KUKA KRL program: ps_a_stb_res_c02.src, ps_a_stb_res_c02.dat

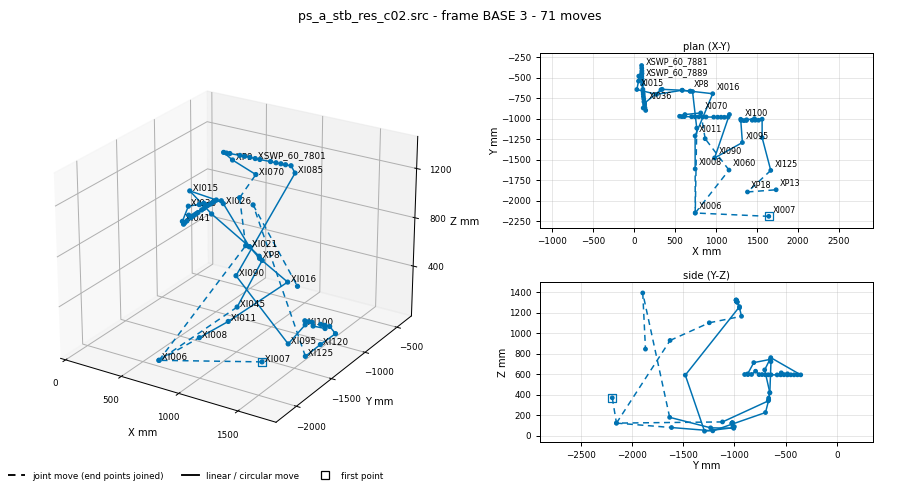
[picture p0: tool path of ps_a_stb_res_c02.src in frame BASE 3, 71 of 71 moves have a stored position in this frame; points joined in program order, loops and branches not executed]
--- ps_a_stb_res_c02.src ---
&ACCESS RVO1
&REL 230
&COMMENT Solda Atego STB
&PARAM DISKPATH = KRC:\R1\Program\OLP
DEF ps_a_stb_res_c02( )

;FOLD INI
;FOLD SPOTTECH INI
USERSPOT(#INIT)
;ENDFOLD (SPOTTECH INI)
;FOLD GRIPPERTECH INI
USER_GRP(0,DUMMY,DUMMY,GDEFAULT)
;ENDFOLD (GRIPPERTECH INI)
  ;FOLD USER INI
    ;Make your modifications here

  ;ENDFOLD (USER INI)
;ENDFOLD (INI)

; Caracterizacao dos meios de producao
; Changes: Solda Respot - ATEGO - STB
; Versao Atual: 18/02/2016
; Ferramenta: Gun C02
; Name: P13.060-R1

chk_w3_wechs_ok ( )              ; CHECK C2

IF (NOT(GHOST())) THEN
IF MaxStandMenge(3) THEN
  MaxStandmengeErreicht(3)
ENDIF
IF Elektrodenwechsel(3) THEN
  e_Fraes_3 ()
ENDIF
ENDIF

;FOLD PTP l007 Vel=100 % P_OLP7 Tool[3]:GUN C2 Base[3]:Atego/Axor;%{PE}%R 8.2.20,%MKUKATPBASIS,%CMOVE,%VPTP,%P 1:PTP, 2:l007, 3:, 5:100, 7:P_OLP7
$BWDSTART=FALSE
PDAT_ACT=PP_OLP7
FDAT_ACT=Fl007
BAS(#PTP_PARAMS,100)
PTP Xl007
;ENDFOLD
;FOLD PTP l006 Vel=100 % P_OLP6 Tool[3]:Gun C02 Base[3]:Atego/Axor;%{PE}%R 8.2.20,%MKUKATPBASIS,%CMOVE,%VPTP,%P 1:PTP, 2:l006, 3:, 5:100, 7:P_OLP6
$BWDSTART=FALSE
PDAT_ACT=PP_OLP6
FDAT_ACT=Fl006
BAS(#PTP_PARAMS,100)
PTP Xl006
;ENDFOLD

;FOLD OUT 3380 'Perfil Livre Estacao' State=TRUE ;%{PE}%R 8.2.20,%MKUKATPBASIS,%COUT,%VOUTX,%P 2:3380, 3:Perfil Livre Estacao, 5:TRUE, 6:
$OUT[3380]=TRUE
;ENDFOLD
;FOLD WAIT FOR ( IN 3380 'Liberacao de Solda' );%{PE}%R 8.2.20,%MKUKATPBASIS,%CEXT_WAIT_FOR,%VEXT_WAIT_FOR,%P 2:, 4:, 5:$IN, 6:3380, 7:Liberacao de Solda, 9:
WAIT FOR  ( $IN[3380] )
;ENDFOLD
;FOLD OUT 3380 'Perfil Livre Estacao' State=FALSE ;%{PE}%R 8.2.20,%MKUKATPBASIS,%COUT,%VOUTX,%P 2:3380, 3:Perfil Livre Estacao, 5:FALSE, 6:
$OUT[3380]=FALSE
;ENDFOLD

;FOLD ; Liga intertravamento 4 com R4;%{PE}%R 8.2.20,%MKUKATPBASIS,%CCOMMENT,%VNORMAL,%P 2:Liga  intertravamento  4  com  R4
;ENDFOLD
;FOLD Collision.Monitoring_4_On ;%{PE}%MKUKATPUSER
COLLSTOP( 4, 1 ) ;Interrupt-Controlled
;ENDFOLD

;FOLD ; Liga intertravamento 10 com R3;%{PE}%R 8.2.20,%MKUKATPBASIS,%CCOMMENT,%VNORMAL,%P 2:Liga  intertravamento  10  com  R3
;ENDFOLD
;FOLD Collision.Monitoring_10_On ;%{PE}%MKUKATPUSER
COLLSTOP( 10, 1 ) ;not Interrupt-Controlled
;ENDFOLD

;FOLD ; Liga intertravamento 5 com R5;%{PE}%R 8.2.20,%MKUKATPBASIS,%CCOMMENT,%VNORMAL,%P 2:Liga  intertravamento  5  com  R5
;ENDFOLD
;FOLD Collision.Monitoring_5_On ;%{PE}%MKUKATPUSER
COLLSTOP( 5, 1 ) ;not Interrupt-Controlled
;ENDFOLD

;FOLD ; Liga intertravamento 12 com R5;%{PE}%R 8.2.20,%MKUKATPBASIS,%CCOMMENT,%VNORMAL,%P 2:Liga  intertravamento  12  com  R5
;ENDFOLD
;FOLD Collision.Monitoring_12_On ;%{PE}%MKUKATPUSER
COLLSTOP( 12, 1 ) ;not Interrupt-Controlled
;ENDFOLD

;FOLD ; Liga intertravamento 13 com R5;%{PE}%R 8.2.20,%MKUKATPBASIS,%CCOMMENT,%VNORMAL,%P 2:Liga  intertravamento  13  com  R5
;ENDFOLD
;FOLD Collision.Monitoring_13_On ;%{PE}%MKUKATPUSER
COLLSTOP( 13, 1 ) ;not Interrupt-Controlled
;ENDFOLD

;FOLD PTP l008 CONT Vel=100 % P_OLP8 Tool[3]:GUN C2 Base[3]:Atego/Axor;%{PE}%R 8.2.20,%MKUKATPBASIS,%CMOVE,%VPTP,%P 1:PTP, 2:l008, 3:C_DIS, 5:100, 7:P_OLP8
$BWDSTART=FALSE
PDAT_ACT=PP_OLP8
FDAT_ACT=Fl008
BAS(#PTP_PARAMS,100)
PTP Xl008 C_DIS
;ENDFOLD
;FOLD LIN l011 CONT Vel=2 m/s L_OLP42 Tool[3]:GUN C2 Base[3]:Atego/Axor;%{PE}%R 8.2.20,%MKUKATPBASIS,%CMOVE,%VLIN,%P 1:LIN, 2:l011, 3:C_DIS C_DIS, 5:2, 7:L_OLP42
$BWDSTART=FALSE
LDAT_ACT=LL_OLP42
FDAT_ACT=Fl011
BAS(#CP_PARAMS,2)
LIN Xl011 C_DIS C_DIS
;ENDFOLD
;FOLD LIN l016 CONT Vel=2 m/s CPDAT11 Tool[3]:GUN C2 Base[3]:Atego/Axor;%{PE}%R 8.2.20,%MKUKATPBASIS,%CMOVE,%VLIN,%P 1:LIN, 2:l016, 3:C_DIS C_DIS, 5:2, 7:CPDAT11
$BWDSTART=FALSE
LDAT_ACT=LCPDAT11
FDAT_ACT=Fl016
BAS(#CP_PARAMS,2)
LIN Xl016 C_DIS C_DIS
;ENDFOLD
;FOLD LIN P8 CONT Vel=2 m/s CPDAT8 Tool[3]:GUN C2 Base[3]:Atego/Axor;%{PE}%R 8.2.20,%MKUKATPBASIS,%CMOVE,%VLIN,%P 1:LIN, 2:P8, 3:C_DIS C_DIS, 5:2, 7:CPDAT8
$BWDSTART=FALSE
LDAT_ACT=LCPDAT8
FDAT_ACT=FP8
BAS(#CP_PARAMS,2)
LIN XP8 C_DIS C_DIS
;ENDFOLD
;FOLD LIN l021 CONT Vel=2 m/s L_OLP44 Tool[3]:GUN C2 Base[3]:Atego/Axor;%{PE}%R 8.2.20,%MKUKATPBASIS,%CMOVE,%VLIN,%P 1:LIN, 2:l021, 3:C_DIS C_DIS, 5:2, 7:L_OLP44
$BWDSTART=FALSE
LDAT_ACT=LL_OLP44
FDAT_ACT=Fl021
BAS(#CP_PARAMS,2)
LIN Xl021 C_DIS C_DIS
;ENDFOLD
;FOLD LIN l026 CONT Vel=2 m/s L_OLP45 Tool[3]:GUN C2 Base[3]:Atego/Axor;%{PE}%R 8.2.20,%MKUKATPBASIS,%CMOVE,%VLIN,%P 1:LIN, 2:l026, 3:C_DIS C_DIS, 5:2, 7:L_OLP45
$BWDSTART=FALSE
LDAT_ACT=LL_OLP45
FDAT_ACT=Fl026
BAS(#CP_PARAMS,2)
LIN Xl026 C_DIS C_DIS
;ENDFOLD
;FOLD LIN l031 CONT Vel=1 m/s L_OLP46 Tool[3]:GUN C2 Base[3]:Atego/Axor;%{PE}%R 8.2.20,%MKUKATPBASIS,%CMOVE,%VLIN,%P 1:LIN, 2:l031, 3:C_DIS C_DIS, 5:1, 7:L_OLP46
$BWDSTART=FALSE
LDAT_ACT=LL_OLP46
FDAT_ACT=Fl031
BAS(#CP_PARAMS,1)
LIN Xl031 C_DIS C_DIS
;ENDFOLD
;FOLD LIN l036 CONT Vel=2 m/s L_OLP47 Tool[3]:GUN C2 Base[3]:Atego/Axor;%{PE}%R 8.2.20,%MKUKATPBASIS,%CMOVE,%VLIN,%P 1:LIN, 2:l036, 3:C_DIS C_DIS, 5:2, 7:L_OLP47
$BWDSTART=FALSE
LDAT_ACT=LL_OLP47
FDAT_ACT=Fl036
BAS(#CP_PARAMS,2)
LIN Xl036 C_DIS C_DIS
;ENDFOLD
;FOLD LIN l041 CONT Vel=2 m/s L_OLP48 Tool[3]:GUN C2 Base[3]:Atego/Axor;%{PE}%R 8.2.20,%MKUKATPBASIS,%CMOVE,%VLIN,%P 1:LIN, 2:l041, 3:C_DIS C_DIS, 5:2, 7:L_OLP48
$BWDSTART=FALSE
LDAT_ACT=LL_OLP48
FDAT_ACT=Fl041
BAS(#CP_PARAMS,2)
LIN Xl041 C_DIS C_DIS
;ENDFOLD

;FOLD ; SWP_60_7345;%{PE}%R 8.2.20,%MKUKATPBASIS,%CCOMMENT,%VNORMAL,%P 2:SWP_60_7345
;ENDFOLD
;FOLD LIN swp_60_7345 CPDAT13 SPOT Gun=2 RETR CLS PgNo1=186 ACTIVE=1 Tool[3]:GUN C2 Base[3]:Atego/Axor;%{PE}%R 8.2.2,%MKUKATPSPOT,%CSPOT,%VLIN,%P 1:LIN, 2:swp_60_7345, 3:, 5:2, 7:CPDAT13, 10:2, 12:#FIRST, 14:#CLO, 16:186, 18:1, 20:0, 22:0, 24:1, 25:NORMAL
$BWDSTART=FALSE
LDAT_ACT=LCPDAT13
FDAT_ACT=Fswp_60_7345
BAS(#CP_PARAMS,LCPDAT13.VEL)
S_ACT.GUN=2
S_ACT.PAIR=SDEFAULT.PAIR
S_ACT.RETR=#CLO
S_ACT.CLO_TM=1
S_ACT.PGNO1=186
S_ACT.PGNO2=SDEFAULT.PGNO2
S_ACT.PRESS1=SDEFAULT.PRESS1
S_ACT.PRESS2=SDEFAULT.PRESS2
S_READY=FALSE
LIN Xswp_60_7345
USERSPOT(#SPOT, S_ACT)
WAIT FOR S_READY
;ENDFOLD

;FOLD ; SWP_60_7909;%{PE}%R 8.2.20,%MKUKATPBASIS,%CCOMMENT,%VNORMAL,%P 2:SWP_60_7909
;ENDFOLD
;FOLD LIN SWP_60_7909 L_OLP49 SPOT Gun=2 RETR CLS PgNo1=186 ACTIVE=1 Tool[3]:GUN C2 Base[3]:Atego/Axor;%{PE}%R 8.2.2,%MKUKATPSPOT,%CSPOT,%VLIN,%P 1:LIN, 2:SWP_60_7909, 3:, 5:2, 7:L_OLP49, 10:2, 12:#FIRST, 14:#CLO, 16:186, 18:1, 20:0, 22:0, 24:1, 25:NORMAL
$BWDSTART=FALSE
LDAT_ACT=LL_OLP49
FDAT_ACT=FSWP_60_7909
BAS(#CP_PARAMS,LL_OLP49.VEL)
S_ACT.GUN=2
S_ACT.PAIR=SDEFAULT.PAIR
S_ACT.RETR=#CLO
S_ACT.CLO_TM=1
S_ACT.PGNO1=186
S_ACT.PGNO2=SDEFAULT.PGNO2
S_ACT.PRESS1=SDEFAULT.PRESS1
S_ACT.PRESS2=SDEFAULT.PRESS2
S_READY=FALSE
LIN XSWP_60_7909
USERSPOT(#SPOT, S_ACT)
WAIT FOR S_READY
;ENDFOLD

;FOLD ; SWP_60_7907;%{PE}%R 8.2.20,%MKUKATPBASIS,%CCOMMENT,%VNORMAL,%P 2:SWP_60_7907
;ENDFOLD
;FOLD LIN SWP_60_7907 CPDAT1 SPOT Gun=2 RETR CLS PgNo1=186 ACTIVE=1 Tool[3]:GUN C2 Base[3]:Atego/Axor;%{PE}%R 8.2.2,%MKUKATPSPOT,%CSPOT,%VLIN,%P 1:LIN, 2:SWP_60_7907, 3:, 5:0.001, 7:CPDAT1, 10:2, 12:#FIRST, 14:#CLO, 16:186, 18:1, 20:0, 22:0, 24:1, 25:NORMAL
$BWDSTART=FALSE
LDAT_ACT=LCPDAT1
FDAT_ACT=FSWP_60_7907
BAS(#CP_PARAMS,LCPDAT1.VEL)
S_ACT.GUN=2
S_ACT.PAIR=SDEFAULT.PAIR
S_ACT.RETR=#CLO
S_ACT.CLO_TM=1
S_ACT.PGNO1=186
S_ACT.PGNO2=SDEFAULT.PGNO2
S_ACT.PRESS1=SDEFAULT.PRESS1
S_ACT.PRESS2=SDEFAULT.PRESS2
S_READY=FALSE
LIN XSWP_60_7907
USERSPOT(#SPOT, S_ACT)
WAIT FOR S_READY
;ENDFOLD

;FOLD LIN l042 CONT Vel=2 m/s L_OLP65 Tool[3]:GUN C2 Base[3]:Atego/Axor;%{PE}%R 8.2.20,%MKUKATPBASIS,%CMOVE,%VLIN,%P 1:LIN, 2:l042, 3:C_DIS C_DIS, 5:2, 7:L_OLP65
$BWDSTART=FALSE
LDAT_ACT=LL_OLP65
FDAT_ACT=Fl042
BAS(#CP_PARAMS,2)
LIN Xl042 C_DIS C_DIS
;ENDFOLD

;FOLD ; SWP_60_7905;%{PE}%R 8.2.20,%MKUKATPBASIS,%CCOMMENT,%VNORMAL,%P 2:SWP_60_7905
;ENDFOLD
;FOLD LIN SWP_60_7905 L_OLP51 SPOT Gun=2 RETR CLS PgNo1=186 ACTIVE=1 Tool[3]:GUN C2 Base[3]:Atego/Axor;%{PE}%R 8.2.2,%MKUKATPSPOT,%CSPOT,%VLIN,%P 1:LIN, 2:SWP_60_7905, 3:, 5:2, 7:L_OLP51, 10:2, 12:#FIRST, 14:#CLO, 16:186, 18:1, 20:0, 22:0, 24:1, 25:NORMAL
$BWDSTART=FALSE
LDAT_ACT=LL_OLP51
FDAT_ACT=FSWP_60_7905
BAS(#CP_PARAMS,LL_OLP51.VEL)
S_ACT.GUN=2
S_ACT.PAIR=SDEFAULT.PAIR
S_ACT.RETR=#CLO
S_ACT.CLO_TM=1
S_ACT.PGNO1=186
S_ACT.PGNO2=SDEFAULT.PGNO2
S_ACT.PRESS1=SDEFAULT.PRESS1
S_ACT.PRESS2=SDEFAULT.PRESS2
S_READY=FALSE
LIN XSWP_60_7905
USERSPOT(#SPOT, S_ACT)
WAIT FOR S_READY
;ENDFOLD

;FOLD ; SWP_60_7903;%{PE}%R 8.2.20,%MKUKATPBASIS,%CCOMMENT,%VNORMAL,%P 2:SWP_60_7903
;ENDFOLD
;FOLD LIN SWP_60_7903 L_OLP52 SPOT Gun=2 RETR CLS PgNo1=186 ACTIVE=1 Tool[3]:GUN C2 Base[3]:Atego/Axor;%{PE}%R 8.2.2,%MKUKATPSPOT,%CSPOT,%VLIN,%P 1:LIN, 2:SWP_60_7903, 3:, 5:2, 7:L_OLP52, 10:2, 12:#FIRST, 14:#CLO, 16:186, 18:1, 20:0, 22:0, 24:1, 25:NORMAL
$BWDSTART=FALSE
LDAT_ACT=LL_OLP52
FDAT_ACT=FSWP_60_7903
BAS(#CP_PARAMS,LL_OLP52.VEL)
S_ACT.GUN=2
S_ACT.PAIR=SDEFAULT.PAIR
S_ACT.RETR=#CLO
S_ACT.CLO_TM=1
S_ACT.PGNO1=186
S_ACT.PGNO2=SDEFAULT.PGNO2
S_ACT.PRESS1=SDEFAULT.PRESS1
S_ACT.PRESS2=SDEFAULT.PRESS2
S_READY=FALSE
LIN XSWP_60_7903
USERSPOT(#SPOT, S_ACT)
WAIT FOR S_READY
;ENDFOLD

;FOLD ; SWP_60_7901;%{PE}%R 8.2.20,%MKUKATPBASIS,%CCOMMENT,%VNORMAL,%P 2:SWP_60_7901
;ENDFOLD
;FOLD LIN SWP_60_7901 L_OLP53 SPOT Gun=2 RETR CLS PgNo1=186 ACTIVE=1 Tool[3]:GUN C2 Base[3]:Atego/Axor;%{PE}%R 8.2.2,%MKUKATPSPOT,%CSPOT,%VLIN,%P 1:LIN, 2:SWP_60_7901, 3:, 5:2, 7:L_OLP53, 10:2, 12:#FIRST, 14:#CLO, 16:186, 18:1, 20:0, 22:0, 24:1, 25:NORMAL
$BWDSTART=FALSE
LDAT_ACT=LL_OLP53
FDAT_ACT=FSWP_60_7901
BAS(#CP_PARAMS,LL_OLP53.VEL)
S_ACT.GUN=2
S_ACT.PAIR=SDEFAULT.PAIR
S_ACT.RETR=#CLO
S_ACT.CLO_TM=1
S_ACT.PGNO1=186
S_ACT.PGNO2=SDEFAULT.PGNO2
S_ACT.PRESS1=SDEFAULT.PRESS1
S_ACT.PRESS2=SDEFAULT.PRESS2
S_READY=FALSE
LIN XSWP_60_7901
USERSPOT(#SPOT, S_ACT)
WAIT FOR S_READY
;ENDFOLD

;FOLD ; SWP_60_7329;%{PE}%R 8.2.20,%MKUKATPBASIS,%CCOMMENT,%VNORMAL,%P 2:SWP_60_7329
;ENDFOLD
;FOLD LIN SWP_60_7329 L_OLP54 SPOT Gun=2 RETR CLS PgNo1=186 ACTIVE=1 Tool[3]:GUN C2 Base[3]:Atego/Axor;%{PE}%R 8.2.2,%MKUKATPSPOT,%CSPOT,%VLIN,%P 1:LIN, 2:SWP_60_7329, 3:, 5:2, 7:L_OLP54, 10:2, 12:#FIRST, 14:#CLO, 16:186, 18:1, 20:0, 22:0, 24:1, 25:NORMAL
$BWDSTART=FALSE
LDAT_ACT=LL_OLP54
FDAT_ACT=FSWP_60_7329
BAS(#CP_PARAMS,LL_OLP54.VEL)
S_ACT.GUN=2
S_ACT.PAIR=SDEFAULT.PAIR
S_ACT.RETR=#CLO
S_ACT.CLO_TM=1
S_ACT.PGNO1=186
S_ACT.PGNO2=SDEFAULT.PGNO2
S_ACT.PRESS1=SDEFAULT.PRESS1
S_ACT.PRESS2=SDEFAULT.PRESS2
S_READY=FALSE
LIN XSWP_60_7329
USERSPOT(#SPOT, S_ACT)
WAIT FOR S_READY
;ENDFOLD

;FOLD ; SWP_60_7897;%{PE}%R 8.2.20,%MKUKATPBASIS,%CCOMMENT,%VNORMAL,%P 2:SWP_60_7897
;ENDFOLD
;FOLD LIN SWP_60_7897 CPDAT14 SPOT Gun=2 RETR CLS PgNo1=186 ACTIVE=1 Tool[3]:GUN C2 Base[3]:Atego/Axor;%{PE}%R 8.2.2,%MKUKATPSPOT,%CSPOT,%VLIN,%P 1:LIN, 2:SWP_60_7897, 3:, 5:2, 7:CPDAT14, 10:2, 12:#FIRST, 14:#CLO, 16:186, 18:1, 20:0, 22:0, 24:1, 25:NORMAL
$BWDSTART=FALSE
LDAT_ACT=LCPDAT14
FDAT_ACT=FSWP_60_7897
BAS(#CP_PARAMS,LCPDAT14.VEL)
S_ACT.GUN=2
S_ACT.PAIR=SDEFAULT.PAIR
S_ACT.RETR=#CLO
S_ACT.CLO_TM=1
S_ACT.PGNO1=186
S_ACT.PGNO2=SDEFAULT.PGNO2
S_ACT.PRESS1=SDEFAULT.PRESS1
S_ACT.PRESS2=SDEFAULT.PRESS2
S_READY=FALSE
LIN XSWP_60_7897
USERSPOT(#SPOT, S_ACT)
WAIT FOR S_READY
;ENDFOLD

;FOLD ; SWP_60_7893;%{PE}%R 8.2.20,%MKUKATPBASIS,%CCOMMENT,%VNORMAL,%P 2:SWP_60_7893
;ENDFOLD
;FOLD LIN SWP_60_7893 L_OLP55 SPOT Gun=2 RETR CLS PgNo1=186 ACTIVE=1 Tool[3]:GUN C2 Base[3]:Atego/Axor;%{PE}%R 8.2.2,%MKUKATPSPOT,%CSPOT,%VLIN,%P 1:LIN, 2:SWP_60_7893, 3:, 5:2, 7:L_OLP55, 10:2, 12:#FIRST, 14:#CLO, 16:186, 18:1, 20:0, 22:0, 24:1, 25:NORMAL
$BWDSTART=FALSE
LDAT_ACT=LL_OLP55
FDAT_ACT=FSWP_60_7893
BAS(#CP_PARAMS,LL_OLP55.VEL)
S_ACT.GUN=2
S_ACT.PAIR=SDEFAULT.PAIR
S_ACT.RETR=#CLO
S_ACT.CLO_TM=1
S_ACT.PGNO1=186
S_ACT.PGNO2=SDEFAULT.PGNO2
S_ACT.PRESS1=SDEFAULT.PRESS1
S_ACT.PRESS2=SDEFAULT.PRESS2
S_READY=FALSE
LIN XSWP_60_7893
USERSPOT(#SPOT, S_ACT)
WAIT FOR S_READY
;ENDFOLD

;FOLD ; SWP_60_7891;%{PE}%R 8.2.20,%MKUKATPBASIS,%CCOMMENT,%VNORMAL,%P 2:SWP_60_7891
;ENDFOLD
;FOLD LIN SWP_60_7891 L_OLP56 SPOT Gun=2 RETR CLS PgNo1=186 ACTIVE=1 Tool[3]:GUN C2 Base[3]:Atego/Axor;%{PE}%R 8.2.2,%MKUKATPSPOT,%CSPOT,%VLIN,%P 1:LIN, 2:SWP_60_7891, 3:, 5:2, 7:L_OLP56, 10:2, 12:#FIRST, 14:#CLO, 16:186, 18:1, 20:0, 22:0, 24:1, 25:NORMAL
$BWDSTART=FALSE
LDAT_ACT=LL_OLP56
FDAT_ACT=FSWP_60_7891
BAS(#CP_PARAMS,LL_OLP56.VEL)
S_ACT.GUN=2
S_ACT.PAIR=SDEFAULT.PAIR
S_ACT.RETR=#CLO
S_ACT.CLO_TM=1
S_ACT.PGNO1=186
S_ACT.PGNO2=SDEFAULT.PGNO2
S_ACT.PRESS1=SDEFAULT.PRESS1
S_ACT.PRESS2=SDEFAULT.PRESS2
S_READY=FALSE
LIN XSWP_60_7891
USERSPOT(#SPOT, S_ACT)
WAIT FOR S_READY
;ENDFOLD

;FOLD ; SWP_60_7889;%{PE}%R 8.2.20,%MKUKATPBASIS,%CCOMMENT,%VNORMAL,%P 2:SWP_60_7889
;ENDFOLD
;FOLD LIN SWP_60_7889 L_OLP57 SPOT Gun=2 RETR OPN PgNo1=186 ACTIVE=1 Tool[3]:GUN C2 Base[3]:Atego/Axor;%{PE}%R 8.2.2,%MKUKATPSPOT,%CSPOT,%VLIN,%P 1:LIN, 2:SWP_60_7889, 3:, 5:2, 7:L_OLP57, 10:2, 12:#FIRST, 14:#OPN, 16:186, 18:1, 20:0, 22:0, 24:1, 25:NORMAL
$BWDSTART=FALSE
LDAT_ACT=LL_OLP57
FDAT_ACT=FSWP_60_7889
BAS(#CP_PARAMS,LL_OLP57.VEL)
S_ACT.GUN=2
S_ACT.PAIR=SDEFAULT.PAIR
S_ACT.RETR=#OPN
S_ACT.CLO_TM=1
S_ACT.PGNO1=186
S_ACT.PGNO2=SDEFAULT.PGNO2
S_ACT.PRESS1=SDEFAULT.PRESS1
S_ACT.PRESS2=SDEFAULT.PRESS2
S_READY=FALSE
LIN XSWP_60_7889
USERSPOT(#SPOT, S_ACT)
WAIT FOR S_READY
;ENDFOLD

;FOLD LIN P4 CONT Vel=1 m/s CPDAT4 Tool[3]:GUN C2 Base[3]:Atego/Axor;%{PE}%R 8.2.20,%MKUKATPBASIS,%CMOVE,%VLIN,%P 1:LIN, 2:P4, 3:C_DIS C_DIS, 5:1, 7:CPDAT4
$BWDSTART=FALSE
LDAT_ACT=LCPDAT4
FDAT_ACT=FP4
BAS(#CP_PARAMS,1)
LIN XP4 C_DIS C_DIS
;ENDFOLD
;FOLD LIN P5 CONT Vel=1 m/s CPDAT5 Tool[3]:GUN C2 Base[3]:Atego/Axor;%{PE}%R 8.2.20,%MKUKATPBASIS,%CMOVE,%VLIN,%P 1:LIN, 2:P5, 3:C_DIS C_DIS, 5:1, 7:CPDAT5
$BWDSTART=FALSE
LDAT_ACT=LCPDAT5
FDAT_ACT=FP5
BAS(#CP_PARAMS,1)
LIN XP5 C_DIS C_DIS
;ENDFOLD

;FOLD ; SWP_60_7887;%{PE}%R 8.2.20,%MKUKATPBASIS,%CCOMMENT,%VNORMAL,%P 2:SWP_60_7887
;ENDFOLD
;FOLD LIN SWP_60_7887 L_OLP58 SPOT Gun=2 RETR CLS PgNo1=186 ACTIVE=1 Tool[3]:GUN C2 Base[3]:Atego/Axor;%{PE}%R 8.2.2,%MKUKATPSPOT,%CSPOT,%VLIN,%P 1:LIN, 2:SWP_60_7887, 3:, 5:2, 7:L_OLP58, 10:2, 12:#FIRST, 14:#CLO, 16:186, 18:1, 20:0, 22:0, 24:1, 25:NORMAL
$BWDSTART=FALSE
LDAT_ACT=LL_OLP58
FDAT_ACT=FSWP_60_7887
BAS(#CP_PARAMS,LL_OLP58.VEL)
S_ACT.GUN=2
S_ACT.PAIR=SDEFAULT.PAIR
S_ACT.RETR=#CLO
S_ACT.CLO_TM=1
S_ACT.PGNO1=186
S_ACT.PGNO2=SDEFAULT.PGNO2
S_ACT.PRESS1=SDEFAULT.PRESS1
S_ACT.PRESS2=SDEFAULT.PRESS2
S_READY=FALSE
LIN XSWP_60_7887
USERSPOT(#SPOT, S_ACT)
WAIT FOR S_READY
;ENDFOLD

;FOLD ; SWP_60_7885;%{PE}%R 8.2.20,%MKUKATPBASIS,%CCOMMENT,%VNORMAL,%P 2:SWP_60_7885
;ENDFOLD
;FOLD LIN SWP_60_7885 L_OLP59 SPOT Gun=2 RETR CLS PgNo1=186 ACTIVE=1 Tool[3]:GUN C2 Base[3]:Atego/Axor;%{PE}%R 8.2.2,%MKUKATPSPOT,%CSPOT,%VLIN,%P 1:LIN, 2:SWP_60_7885, 3:, 5:2, 7:L_OLP59, 10:2, 12:#FIRST, 14:#CLO, 16:186, 18:1, 20:0, 22:0, 24:1, 25:NORMAL
$BWDSTART=FALSE
LDAT_ACT=LL_OLP59
FDAT_ACT=FSWP_60_7885
BAS(#CP_PARAMS,LL_OLP59.VEL)
S_ACT.GUN=2
S_ACT.PAIR=SDEFAULT.PAIR
S_ACT.RETR=#CLO
S_ACT.CLO_TM=1
S_ACT.PGNO1=186
S_ACT.PGNO2=SDEFAULT.PGNO2
S_ACT.PRESS1=SDEFAULT.PRESS1
S_ACT.PRESS2=SDEFAULT.PRESS2
S_READY=FALSE
LIN XSWP_60_7885
USERSPOT(#SPOT, S_ACT)
WAIT FOR S_READY
;ENDFOLD

;FOLD ; SWP_60_7883;%{PE}%R 8.2.20,%MKUKATPBASIS,%CCOMMENT,%VNORMAL,%P 2:SWP_60_7883
;ENDFOLD
;FOLD LIN SWP_60_7883 L_OLP60 SPOT Gun=2 RETR CLS PgNo1=186 ACTIVE=1 Tool[3]:GUN C2 Base[3]:Atego/Axor;%{PE}%R 8.2.2,%MKUKATPSPOT,%CSPOT,%VLIN,%P 1:LIN, 2:SWP_60_7883, 3:, 5:2, 7:L_OLP60, 10:2, 12:#FIRST, 14:#CLO, 16:186, 18:1, 20:0, 22:0, 24:1, 25:NORMAL
$BWDSTART=FALSE
LDAT_ACT=LL_OLP60
FDAT_ACT=FSWP_60_7883
BAS(#CP_PARAMS,LL_OLP60.VEL)
S_ACT.GUN=2
S_ACT.PAIR=SDEFAULT.PAIR
S_ACT.RETR=#CLO
S_ACT.CLO_TM=1
S_ACT.PGNO1=186
S_ACT.PGNO2=SDEFAULT.PGNO2
S_ACT.PRESS1=SDEFAULT.PRESS1
S_ACT.PRESS2=SDEFAULT.PRESS2
S_READY=FALSE
LIN XSWP_60_7883
USERSPOT(#SPOT, S_ACT)
WAIT FOR S_READY
;ENDFOLD

;FOLD ; SWP_60_7881;%{PE}%R 8.2.20,%MKUKATPBASIS,%CCOMMENT,%VNORMAL,%P 2:SWP_60_7881
;ENDFOLD
;FOLD LIN SWP_60_7881 L_OLP61 SPOT Gun=2 RETR CLS PgNo1=186 ACTIVE=1 Tool[3]:GUN C2 Base[3]:Atego/Axor;%{PE}%R 8.2.2,%MKUKATPSPOT,%CSPOT,%VLIN,%P 1:LIN, 2:SWP_60_7881, 3:, 5:2, 7:L_OLP61, 10:2, 12:#FIRST, 14:#CLO, 16:186, 18:1, 20:0, 22:0, 24:1, 25:NORMAL
$BWDSTART=FALSE
LDAT_ACT=LL_OLP61
FDAT_ACT=FSWP_60_7881
BAS(#CP_PARAMS,LL_OLP61.VEL)
S_ACT.GUN=2
S_ACT.PAIR=SDEFAULT.PAIR
S_ACT.RETR=#CLO
S_ACT.CLO_TM=1
S_ACT.PGNO1=186
S_ACT.PGNO2=SDEFAULT.PGNO2
S_ACT.PRESS1=SDEFAULT.PRESS1
S_ACT.PRESS2=SDEFAULT.PRESS2
S_READY=FALSE
LIN XSWP_60_7881
USERSPOT(#SPOT, S_ACT)
WAIT FOR S_READY
;ENDFOLD

;FOLD ; SWP_60_7311;%{PE}%R 8.2.20,%MKUKATPBASIS,%CCOMMENT,%VNORMAL,%P 2:SWP_60_7311
;ENDFOLD
;FOLD LIN SWP_60_7311 L_OLP48 SPOT Gun=2 RETR CLS PgNo1=186 ACTIVE=1 Tool[3]:GUN C2 Base[3]:Atego/Axor;%{PE}%R 8.2.2,%MKUKATPSPOT,%CSPOT,%VLIN,%P 1:LIN, 2:SWP_60_7311, 3:, 5:2, 7:L_OLP48, 10:2, 12:#FIRST, 14:#CLO, 16:186, 18:1, 20:0, 22:0, 24:1, 25:NORMAL
$BWDSTART=FALSE
LDAT_ACT=LL_OLP48
FDAT_ACT=FSWP_60_7311
BAS(#CP_PARAMS,LL_OLP48.VEL)
S_ACT.GUN=2
S_ACT.PAIR=SDEFAULT.PAIR
S_ACT.RETR=#CLO
S_ACT.CLO_TM=1
S_ACT.PGNO1=186
S_ACT.PGNO2=SDEFAULT.PGNO2
S_ACT.PRESS1=SDEFAULT.PRESS1
S_ACT.PRESS2=SDEFAULT.PRESS2
S_READY=FALSE
LIN XSWP_60_7311
USERSPOT(#SPOT, S_ACT)
WAIT FOR S_READY
;ENDFOLD

;FOLD LIN l015  Vel=2.00 m/s L_OLP3 Tool[3]:GUN C2 Base[3]:Atego/Axor;%{PE}%R8.2.19,%MKUKATPBASIS,%CMOVE,%VLIN,%P 1:LIN, 2:l015, 3: , 5:2.00, 7:L_OLP3
$BWDSTART = FALSE
LDAT_ACT= LL_OLP3
FDAT_ACT= Fl015
BAS(#CP_PARAMS,2.00)
LIN Xl015
;ENDFOLD
;FOLD LIN l030 CONT Vel=2 m/s L_OLP6 Tool[3]:GUN C2 Base[3]:Atego/Axor;%{PE}%R 8.2.20,%MKUKATPBASIS,%CMOVE,%VLIN,%P 1:LIN, 2:l030, 3:C_DIS C_DIS, 5:2, 7:L_OLP6
$BWDSTART=FALSE
LDAT_ACT=LL_OLP6
FDAT_ACT=Fl030
BAS(#CP_PARAMS,2)
LIN Xl030 C_DIS C_DIS
;ENDFOLD
;FOLD LIN l035 CONT Vel=2 m/s L_OLP7 Tool[3]:GUN C2 Base[3]:Atego/Axor;%{PE}%R 8.2.20,%MKUKATPBASIS,%CMOVE,%VLIN,%P 1:LIN, 2:l035, 3:C_DIS C_DIS, 5:2, 7:L_OLP7
$BWDSTART=FALSE
LDAT_ACT=LL_OLP7
FDAT_ACT=Fl035
BAS(#CP_PARAMS,2)
LIN Xl035 C_DIS C_DIS
;ENDFOLD
;FOLD LIN P7 CONT Vel=2 m/s CPDAT7 Tool[3]:GUN C2 Base[3]:Atego/Axor;%{PE}%R 8.2.20,%MKUKATPBASIS,%CMOVE,%VLIN,%P 1:LIN, 2:P7, 3:C_DIS C_DIS, 5:2, 7:CPDAT7
$BWDSTART=FALSE
LDAT_ACT=LCPDAT7
FDAT_ACT=FP7
BAS(#CP_PARAMS,2)
LIN XP7 C_DIS C_DIS
;ENDFOLD
;FOLD LIN l040 CONT Vel=2 m/s L_OLP8 Tool[3]:GUN C2 Base[3]:Atego/Axor;%{PE}%R 8.2.20,%MKUKATPBASIS,%CMOVE,%VLIN,%P 1:LIN, 2:l040, 3:C_DIS C_DIS, 5:2, 7:L_OLP8
$BWDSTART=FALSE
LDAT_ACT=LL_OLP8
FDAT_ACT=Fl040
BAS(#CP_PARAMS,2)
LIN Xl040 C_DIS C_DIS
;ENDFOLD
;FOLD LIN l045 CONT Vel=2 m/s L_OLP9 Tool[3]:GUN C2 Base[3]:Atego/Axor;%{PE}%R 8.2.20,%MKUKATPBASIS,%CMOVE,%VLIN,%P 1:LIN, 2:l045, 3:C_DIS C_DIS, 5:2, 7:L_OLP9
$BWDSTART=FALSE
LDAT_ACT=LL_OLP9
FDAT_ACT=Fl045
BAS(#CP_PARAMS,2)
LIN Xl045 C_DIS C_DIS
;ENDFOLD
;FOLD PTP l050 Vel=100 % PDAT4 Tool[3]:GUN C2 Base[3]:Atego/Axor;%{PE}%R 8.2.20,%MKUKATPBASIS,%CMOVE,%VPTP,%P 1:PTP, 2:l050, 3:, 5:100, 7:PDAT4
$BWDSTART=FALSE
PDAT_ACT=PPDAT4
FDAT_ACT=Fl050
BAS(#PTP_PARAMS,100)
PTP Xl050
;ENDFOLD

;FOLD ; Desliga intertravamento 4 com R4;%{PE}%R 8.2.20,%MKUKATPBASIS,%CCOMMENT,%VNORMAL,%P 2:Desliga  intertravamento  4  com  R4
;ENDFOLD
;FOLD Collision.Monitoring_4_Off . ;%{PE}%MKUKATPUSER
COLLSTOP( 4, 2+0 )
;ENDFOLD

;FOLD ; Desliga intertravamento 10 com R3;%{PE}%R 8.2.20,%MKUKATPBASIS,%CCOMMENT,%VNORMAL,%P 2:Desliga  intertravamento  10  com  R3
;ENDFOLD
;FOLD Collision.Monitoring_10_Off . ;%{PE}%MKUKATPUSER
COLLSTOP( 10, 2+0 )
;ENDFOLD

;FOLD ; Desliga intertravamento 5 com R5;%{PE}%R 8.2.20,%MKUKATPBASIS,%CCOMMENT,%VNORMAL,%P 2:Desliga  intertravamento  5  com  R5
;ENDFOLD
;FOLD Collision.Monitoring_5_Off . ;%{PE}%MKUKATPUSER
COLLSTOP( 5, 2+0 )
;ENDFOLD

;FOLD ; Desliga intertravamento 13 com R5;%{PE}%R 8.2.20,%MKUKATPBASIS,%CCOMMENT,%VNORMAL,%P 2:Desliga  intertravamento  13  com  R5
;ENDFOLD
;FOLD Collision.Monitoring_13_Off . ;%{PE}%MKUKATPUSER
COLLSTOP( 13, 2+0 )
;ENDFOLD

;FOLD PTP l060 CONT Vel=100 % P_OLP2 Tool[3]:GUN C2 Base[3]:Atego/Axor;%{PE}%R 8.2.20,%MKUKATPBASIS,%CMOVE,%VPTP,%P 1:PTP, 2:l060, 3:C_DIS, 5:100, 7:P_OLP2
$BWDSTART=FALSE
PDAT_ACT=PP_OLP2
FDAT_ACT=Fl060
BAS(#PTP_PARAMS,100)
PTP Xl060 C_DIS
;ENDFOLD
;FOLD PTP l065 CONT Vel=100 % P_OLP3 Tool[3]:GUN C2 Base[3]:Atego/Axor;%{PE}%R 8.2.20,%MKUKATPBASIS,%CMOVE,%VPTP,%P 1:PTP, 2:l065, 3:C_DIS, 5:100, 7:P_OLP3
$BWDSTART=FALSE
PDAT_ACT=PP_OLP3
FDAT_ACT=Fl065
BAS(#PTP_PARAMS,100)
PTP Xl065 C_DIS
;ENDFOLD
;FOLD PTP l070 CONT Vel=100 % P_OLP4 Tool[3]:GUN C2 Base[3]:Atego/Axor;%{PE}%R 8.2.20,%MKUKATPBASIS,%CMOVE,%VPTP,%P 1:PTP, 2:l070, 3:C_DIS, 5:100, 7:P_OLP4
$BWDSTART=FALSE
PDAT_ACT=PP_OLP4
FDAT_ACT=Fl070
BAS(#PTP_PARAMS,100)
PTP Xl070 C_DIS
;ENDFOLD
;FOLD LIN P9 Vel=2 m/s CPDAT9 Tool[3]:GUN C2 Base[3]:Atego/Axor;%{PE}%R 8.2.20,%MKUKATPBASIS,%CMOVE,%VLIN,%P 1:LIN, 2:P9, 3:, 5:2, 7:CPDAT9
$BWDSTART=FALSE
LDAT_ACT=LCPDAT9
FDAT_ACT=FP9
BAS(#CP_PARAMS,2)
LIN XP9
;ENDFOLD

;FOLD ; SWP_60_7787;%{PE}%R 4.1.16,%MKUKATPBASIS,%CCOMMENT,%VNORMAL,%P 2:SWP_60_7787
;ENDFOLD
;FOLD LIN SWP_60_7787 L_OLP12 SPOT Gun=2 RETR CLS PgNo1=184 ACTIVE=1 Tool[3]:GUN C2 Base[3]:Atego/Axor;%{PE}%R 8.2.2,%MKUKATPSPOT,%CSPOT,%VLIN,%P 1:LIN, 2:SWP_60_7787, 3:, 5:2, 7:L_OLP12, 10:2, 12:#FIRST, 14:#CLO, 16:184, 18:1, 20:0, 22:0, 24:1, 25:NORMAL
$BWDSTART=FALSE
LDAT_ACT=LL_OLP12
FDAT_ACT=FSWP_60_7787
BAS(#CP_PARAMS,LL_OLP12.VEL)
S_ACT.GUN=2
S_ACT.PAIR=SDEFAULT.PAIR
S_ACT.RETR=#CLO
S_ACT.CLO_TM=1
S_ACT.PGNO1=184
S_ACT.PGNO2=SDEFAULT.PGNO2
S_ACT.PRESS1=SDEFAULT.PRESS1
S_ACT.PRESS2=SDEFAULT.PRESS2
S_READY=FALSE
LIN XSWP_60_7787
USERSPOT(#SPOT, S_ACT)
WAIT FOR S_READY
;ENDFOLD

;FOLD ; SWP_60_7789;%{PE}%R 4.1.16,%MKUKATPBASIS,%CCOMMENT,%VNORMAL,%P 2:SWP_60_7789
;ENDFOLD
;FOLD LIN SWP_60_7789 L_OLP13 SPOT Gun=2 RETR CLS PgNo1=184 ACTIVE=1 Tool[3]:GUN C2 Base[3]:Atego/Axor;%{PE}%R 8.2.2,%MKUKATPSPOT,%CSPOT,%VLIN,%P 1:LIN, 2:SWP_60_7789, 3:, 5:2, 7:L_OLP13, 10:2, 12:#FIRST, 14:#CLO, 16:184, 18:1, 20:0, 22:0, 24:1, 25:NORMAL
$BWDSTART=FALSE
LDAT_ACT=LL_OLP13
FDAT_ACT=FSWP_60_7789
BAS(#CP_PARAMS,LL_OLP13.VEL)
S_ACT.GUN=2
S_ACT.PAIR=SDEFAULT.PAIR
S_ACT.RETR=#CLO
S_ACT.CLO_TM=1
S_ACT.PGNO1=184
S_ACT.PGNO2=SDEFAULT.PGNO2
S_ACT.PRESS1=SDEFAULT.PRESS1
S_ACT.PRESS2=SDEFAULT.PRESS2
S_READY=FALSE
LIN XSWP_60_7789
USERSPOT(#SPOT, S_ACT)
WAIT FOR S_READY
;ENDFOLD

;FOLD ; SWP_60_7791;%{PE}%R 4.1.16,%MKUKATPBASIS,%CCOMMENT,%VNORMAL,%P 2:SWP_60_7791
;ENDFOLD
;FOLD LIN SWP_60_7791 L_OLP14 SPOT Gun=2 RETR CLS PgNo1=184 ACTIVE=1 Tool[3]:GUN C2 Base[3]:Atego/Axor;%{PE}%R 8.2.2,%MKUKATPSPOT,%CSPOT,%VLIN,%P 1:LIN, 2:SWP_60_7791, 3:, 5:2, 7:L_OLP14, 10:2, 12:#FIRST, 14:#CLO, 16:184, 18:1, 20:0, 22:0, 24:1, 25:NORMAL
$BWDSTART=FALSE
LDAT_ACT=LL_OLP14
FDAT_ACT=FSWP_60_7791
BAS(#CP_PARAMS,LL_OLP14.VEL)
S_ACT.GUN=2
S_ACT.PAIR=SDEFAULT.PAIR
S_ACT.RETR=#CLO
S_ACT.CLO_TM=1
S_ACT.PGNO1=184
S_ACT.PGNO2=SDEFAULT.PGNO2
S_ACT.PRESS1=SDEFAULT.PRESS1
S_ACT.PRESS2=SDEFAULT.PRESS2
S_READY=FALSE
LIN XSWP_60_7791
USERSPOT(#SPOT, S_ACT)
WAIT FOR S_READY
;ENDFOLD

;FOLD ; SWP_60_7795;%{PE}%R 4.1.16,%MKUKATPBASIS,%CCOMMENT,%VNORMAL,%P 2:SWP_60_7795
;ENDFOLD
;FOLD LIN SWP_60_7795 L_OLP16 SPOT Gun=2 RETR CLS PgNo1=182 ACTIVE=1 Tool[3]:GUN C2 Base[3]:Atego/Axor;%{PE}%R 8.2.2,%MKUKATPSPOT,%CSPOT,%VLIN,%P 1:LIN, 2:SWP_60_7795, 3:, 5:2, 7:L_OLP16, 10:2, 12:#FIRST, 14:#CLO, 16:182, 18:1, 20:0, 22:0, 24:1, 25:NORMAL
$BWDSTART=FALSE
LDAT_ACT=LL_OLP16
FDAT_ACT=FSWP_60_7795
BAS(#CP_PARAMS,LL_OLP16.VEL)
S_ACT.GUN=2
S_ACT.PAIR=SDEFAULT.PAIR
S_ACT.RETR=#CLO
S_ACT.CLO_TM=1
S_ACT.PGNO1=182
S_ACT.PGNO2=SDEFAULT.PGNO2
S_ACT.PRESS1=SDEFAULT.PRESS1
S_ACT.PRESS2=SDEFAULT.PRESS2
S_READY=FALSE
LIN XSWP_60_7795
USERSPOT(#SPOT, S_ACT)
WAIT FOR S_READY
;ENDFOLD

;FOLD ; SWP_60_7797;%{PE}%R 4.1.16,%MKUKATPBASIS,%CCOMMENT,%VNORMAL,%P 2:SWP_60_7797
;ENDFOLD
;FOLD LIN SWP_60_7797 L_OLP17 SPOT Gun=2 RETR CLS PgNo1=182 ACTIVE=1 Tool[3]:GUN C2 Base[3]:Atego/Axor;%{PE}%R 8.2.2,%MKUKATPSPOT,%CSPOT,%VLIN,%P 1:LIN, 2:SWP_60_7797, 3:, 5:2, 7:L_OLP17, 10:2, 12:#FIRST, 14:#CLO, 16:182, 18:1, 20:0, 22:0, 24:1, 25:NORMAL
$BWDSTART=FALSE
LDAT_ACT=LL_OLP17
FDAT_ACT=FSWP_60_7797
BAS(#CP_PARAMS,LL_OLP17.VEL)
S_ACT.GUN=2
S_ACT.PAIR=SDEFAULT.PAIR
S_ACT.RETR=#CLO
S_ACT.CLO_TM=1
S_ACT.PGNO1=182
S_ACT.PGNO2=SDEFAULT.PGNO2
S_ACT.PRESS1=SDEFAULT.PRESS1
S_ACT.PRESS2=SDEFAULT.PRESS2
S_READY=FALSE
LIN XSWP_60_7797
USERSPOT(#SPOT, S_ACT)
WAIT FOR S_READY
;ENDFOLD

;FOLD ; SWP_60_7799;%{PE}%R 4.1.16,%MKUKATPBASIS,%CCOMMENT,%VNORMAL,%P 2:SWP_60_7799
;ENDFOLD
;FOLD LIN SWP_60_7799 L_OLP18 SPOT Gun=2 RETR CLS PgNo1=182 ACTIVE=1 Tool[3]:GUN C2 Base[3]:Atego/Axor;%{PE}%R 8.2.2,%MKUKATPSPOT,%CSPOT,%VLIN,%P 1:LIN, 2:SWP_60_7799, 3:, 5:2, 7:L_OLP18, 10:2, 12:#FIRST, 14:#CLO, 16:182, 18:1, 20:0, 22:0, 24:1, 25:NORMAL
$BWDSTART=FALSE
LDAT_ACT=LL_OLP18
FDAT_ACT=FSWP_60_7799
BAS(#CP_PARAMS,LL_OLP18.VEL)
S_ACT.GUN=2
S_ACT.PAIR=SDEFAULT.PAIR
S_ACT.RETR=#CLO
S_ACT.CLO_TM=1
S_ACT.PGNO1=182
S_ACT.PGNO2=SDEFAULT.PGNO2
S_ACT.PRESS1=SDEFAULT.PRESS1
S_ACT.PRESS2=SDEFAULT.PRESS2
S_READY=FALSE
LIN XSWP_60_7799
USERSPOT(#SPOT, S_ACT)
WAIT FOR S_READY
;ENDFOLD

;FOLD ; SWP_60_7801;%{PE}%R 4.1.16,%MKUKATPBASIS,%CCOMMENT,%VNORMAL,%P 2:SWP_60_7801
;ENDFOLD
;FOLD LIN SWP_60_7801 L_OLP19 SPOT Gun=2 RETR CLS PgNo1=182 ACTIVE=1 Tool[3]:GUN C2 Base[3]:Atego/Axor;%{PE}%R 8.2.2,%MKUKATPSPOT,%CSPOT,%VLIN,%P 1:LIN, 2:SWP_60_7801, 3:, 5:2, 7:L_OLP19, 10:2, 12:#FIRST, 14:#CLO, 16:182, 18:1, 20:0, 22:0, 24:1, 25:NORMAL
$BWDSTART=FALSE
LDAT_ACT=LL_OLP19
FDAT_ACT=FSWP_60_7801
BAS(#CP_PARAMS,LL_OLP19.VEL)
S_ACT.GUN=2
S_ACT.PAIR=SDEFAULT.PAIR
S_ACT.RETR=#CLO
S_ACT.CLO_TM=1
S_ACT.PGNO1=182
S_ACT.PGNO2=SDEFAULT.PGNO2
S_ACT.PRESS1=SDEFAULT.PRESS1
S_ACT.PRESS2=SDEFAULT.PRESS2
S_READY=FALSE
LIN XSWP_60_7801
USERSPOT(#SPOT, S_ACT)
WAIT FOR S_READY
;ENDFOLD

;FOLD ; SWP_60_7803;%{PE}%R 4.1.16,%MKUKATPBASIS,%CCOMMENT,%VNORMAL,%P 2:SWP_60_7803
;ENDFOLD
;FOLD LIN SWP_60_7803 L_OLP20 SPOT Gun=2 RETR CLS PgNo1=182 ACTIVE=1 Tool[3]:GUN C2 Base[3]:Atego/Axor;%{PE}%R 8.2.2,%MKUKATPSPOT,%CSPOT,%VLIN,%P 1:LIN, 2:SWP_60_7803, 3:, 5:2, 7:L_OLP20, 10:2, 12:#FIRST, 14:#CLO, 16:182, 18:1, 20:0, 22:0, 24:1, 25:NORMAL
$BWDSTART=FALSE
LDAT_ACT=LL_OLP20
FDAT_ACT=FSWP_60_7803
BAS(#CP_PARAMS,LL_OLP20.VEL)
S_ACT.GUN=2
S_ACT.PAIR=SDEFAULT.PAIR
S_ACT.RETR=#CLO
S_ACT.CLO_TM=1
S_ACT.PGNO1=182
S_ACT.PGNO2=SDEFAULT.PGNO2
S_ACT.PRESS1=SDEFAULT.PRESS1
S_ACT.PRESS2=SDEFAULT.PRESS2
S_READY=FALSE
LIN XSWP_60_7803
USERSPOT(#SPOT, S_ACT)
WAIT FOR S_READY
;ENDFOLD

;FOLD ; SWP_60_7807;%{PE}%R 4.1.16,%MKUKATPBASIS,%CCOMMENT,%VNORMAL,%P 2:SWP_60_7807
;ENDFOLD
;FOLD LIN SWP_60_7807 L_OLP21 SPOT Gun=2 RETR CLS PgNo1=182 ACTIVE=1 Tool[3]:GUN C2 Base[3]:Atego/Axor;%{PE}%R 8.2.2,%MKUKATPSPOT,%CSPOT,%VLIN,%P 1:LIN, 2:SWP_60_7807, 3:, 5:2, 7:L_OLP21, 10:2, 12:#FIRST, 14:#CLO, 16:182, 18:1, 20:0, 22:0, 24:1, 25:NORMAL
$BWDSTART=FALSE
LDAT_ACT=LL_OLP21
FDAT_ACT=FSWP_60_7807
BAS(#CP_PARAMS,LL_OLP21.VEL)
S_ACT.GUN=2
S_ACT.PAIR=SDEFAULT.PAIR
S_ACT.RETR=#CLO
S_ACT.CLO_TM=1
S_ACT.PGNO1=182
S_ACT.PGNO2=SDEFAULT.PGNO2
S_ACT.PRESS1=SDEFAULT.PRESS1
S_ACT.PRESS2=SDEFAULT.PRESS2
S_READY=FALSE
LIN XSWP_60_7807
USERSPOT(#SPOT, S_ACT)
WAIT FOR S_READY
;ENDFOLD

;FOLD ; SWP_60_7809;%{PE}%R 4.1.16,%MKUKATPBASIS,%CCOMMENT,%VNORMAL,%P 2:SWP_60_7809
;ENDFOLD
;FOLD LIN SWP_60_7809 L_OLP22 SPOT Gun=2 RETR CLS PgNo1=182 ACTIVE=1 Tool[3]:GUN C2 Base[3]:Atego/Axor;%{PE}%R 8.2.2,%MKUKATPSPOT,%CSPOT,%VLIN,%P 1:LIN, 2:SWP_60_7809, 3:, 5:2, 7:L_OLP22, 10:2, 12:#FIRST, 14:#CLO, 16:182, 18:1, 20:0, 22:0, 24:1, 25:NORMAL
$BWDSTART=FALSE
LDAT_ACT=LL_OLP22
FDAT_ACT=FSWP_60_7809
BAS(#CP_PARAMS,LL_OLP22.VEL)
S_ACT.GUN=2
S_ACT.PAIR=SDEFAULT.PAIR
S_ACT.RETR=#CLO
S_ACT.CLO_TM=1
S_ACT.PGNO1=182
S_ACT.PGNO2=SDEFAULT.PGNO2
S_ACT.PRESS1=SDEFAULT.PRESS1
S_ACT.PRESS2=SDEFAULT.PRESS2
S_READY=FALSE
LIN XSWP_60_7809
USERSPOT(#SPOT, S_ACT)
WAIT FOR S_READY
;ENDFOLD

;FOLD ; SWP_60_7811;%{PE}%R 4.1.16,%MKUKATPBASIS,%CCOMMENT,%VNORMAL,%P 2:SWP_60_7811
;ENDFOLD
;FOLD LIN SWP_60_7811 L_OLP23 SPOT Gun=2 RETR CLS PgNo1=182 ACTIVE=1 Tool[3]:GUN C2 Base[3]:Atego/Axor;%{PE}%R 8.2.2,%MKUKATPSPOT,%CSPOT,%VLIN,%P 1:LIN, 2:SWP_60_7811, 3:, 5:2, 7:L_OLP23, 10:2, 12:#FIRST, 14:#CLO, 16:182, 18:1, 20:0, 22:0, 24:1, 25:NORMAL
$BWDSTART=FALSE
LDAT_ACT=LL_OLP23
FDAT_ACT=FSWP_60_7811
BAS(#CP_PARAMS,LL_OLP23.VEL)
S_ACT.GUN=2
S_ACT.PAIR=SDEFAULT.PAIR
S_ACT.RETR=#CLO
S_ACT.CLO_TM=1
S_ACT.PGNO1=182
S_ACT.PGNO2=SDEFAULT.PGNO2
S_ACT.PRESS1=SDEFAULT.PRESS1
S_ACT.PRESS2=SDEFAULT.PRESS2
S_READY=FALSE
LIN XSWP_60_7811
USERSPOT(#SPOT, S_ACT)
WAIT FOR S_READY
;ENDFOLD

;FOLD ; SWP_60_7813;%{PE}%R 4.1.16,%MKUKATPBASIS,%CCOMMENT,%VNORMAL,%P 2:SWP_60_7813
;ENDFOLD
;FOLD LIN SWP_60_7813 L_OLP24 SPOT Gun=2 RETR CLS PgNo1=182 ACTIVE=1 Tool[3]:GUN C2 Base[3]:Atego/Axor;%{PE}%R 8.2.2,%MKUKATPSPOT,%CSPOT,%VLIN,%P 1:LIN, 2:SWP_60_7813, 3:, 5:2, 7:L_OLP24, 10:2, 12:#FIRST, 14:#CLO, 16:182, 18:1, 20:0, 22:0, 24:1, 25:NORMAL
$BWDSTART=FALSE
LDAT_ACT=LL_OLP24
FDAT_ACT=FSWP_60_7813
BAS(#CP_PARAMS,LL_OLP24.VEL)
S_ACT.GUN=2
S_ACT.PAIR=SDEFAULT.PAIR
S_ACT.RETR=#CLO
S_ACT.CLO_TM=1
S_ACT.PGNO1=182
S_ACT.PGNO2=SDEFAULT.PGNO2
S_ACT.PRESS1=SDEFAULT.PRESS1
S_ACT.PRESS2=SDEFAULT.PRESS2
S_READY=FALSE
LIN XSWP_60_7813
USERSPOT(#SPOT, S_ACT)
WAIT FOR S_READY
;ENDFOLD

;FOLD ; SWP_60_7815;%{PE}%R 4.1.16,%MKUKATPBASIS,%CCOMMENT,%VNORMAL,%P 2:SWP_60_7815
;ENDFOLD
;FOLD LIN SWP_60_7815 L_OLP25 SPOT Gun=2 RETR OPN PgNo1=182 ACTIVE=1 Tool[3]:GUN C2 Base[3]:Atego/Axor;%{PE}%R 8.2.2,%MKUKATPSPOT,%CSPOT,%VLIN,%P 1:LIN, 2:SWP_60_7815, 3:, 5:2, 7:L_OLP25, 10:2, 12:#FIRST, 14:#OPN, 16:182, 18:1, 20:0, 22:0, 24:1, 25:NORMAL
$BWDSTART=FALSE
LDAT_ACT=LL_OLP25
FDAT_ACT=FSWP_60_7815
BAS(#CP_PARAMS,LL_OLP25.VEL)
S_ACT.GUN=2
S_ACT.PAIR=SDEFAULT.PAIR
S_ACT.RETR=#OPN
S_ACT.CLO_TM=1
S_ACT.PGNO1=182
S_ACT.PGNO2=SDEFAULT.PGNO2
S_ACT.PRESS1=SDEFAULT.PRESS1
S_ACT.PRESS2=SDEFAULT.PRESS2
S_READY=FALSE
LIN XSWP_60_7815
USERSPOT(#SPOT, S_ACT)
WAIT FOR S_READY
;ENDFOLD

;FOLD LIN l085 Vel=2 m/s L_OLP27 Tool[3]:GUN C2 Base[3]:Atego/Axor;%{PE}%R 8.2.20,%MKUKATPBASIS,%CMOVE,%VLIN,%P 1:LIN, 2:l085, 3:, 5:2, 7:L_OLP27
$BWDSTART=FALSE
LDAT_ACT=LL_OLP27
FDAT_ACT=Fl085
BAS(#CP_PARAMS,2)
LIN Xl085
;ENDFOLD
;FOLD LIN l090 Vel=2 m/s L_OLP28 Tool[3]:GUN C2 Base[3]:Atego/Axor;%{PE}%R 8.2.20,%MKUKATPBASIS,%CMOVE,%VLIN,%P 1:LIN, 2:l090, 3:, 5:2, 7:L_OLP28
$BWDSTART=FALSE
LDAT_ACT=LL_OLP28
FDAT_ACT=Fl090
BAS(#CP_PARAMS,2)
LIN Xl090
;ENDFOLD

;FOLD ; Desliga intertravamento 12 com R5;%{PE}%R 8.2.20,%MKUKATPBASIS,%CCOMMENT,%VNORMAL,%P 2:Desliga  intertravamento  12  com  R5
;ENDFOLD
;FOLD Collision.Monitoring_12_Off . ;%{PE}%MKUKATPUSER
COLLSTOP( 12, 2+0 )
;ENDFOLD

;FOLD LIN l095 CONT Vel=2 m/s L_OLP29 Tool[3]:GUN C2 Base[3]:Atego/Axor;%{PE}%R 8.2.20,%MKUKATPBASIS,%CMOVE,%VLIN,%P 1:LIN, 2:l095, 3:C_DIS C_DIS, 5:2, 7:L_OLP29
$BWDSTART=FALSE
LDAT_ACT=LL_OLP29
FDAT_ACT=Fl095
BAS(#CP_PARAMS,2)
LIN Xl095 C_DIS C_DIS
;ENDFOLD
;FOLD LIN l100  Vel=2.00 m/s L_OLP30 Tool[3]:Gun C02 Base[3]:Atego/Axor;%{PE}%R8.2.19,%MKUKATPBASIS,%CMOVE,%VLIN,%P 1:LIN, 2:l100, 3: , 5:2.00, 7:L_OLP30
$BWDSTART = FALSE
LDAT_ACT= LL_OLP30
FDAT_ACT= Fl100
BAS(#CP_PARAMS,2.00)
LIN Xl100
;ENDFOLD

;FOLD ; SWP_60_7487;%{PE}%R 4.1.16,%MKUKATPBASIS,%CCOMMENT,%VNORMAL,%P 2:SWP_60_7487
;ENDFOLD
;FOLD LIN SWP_60_7487 L_OLP31 SPOT Gun=2 RETR CLS PgNo1=185 ACTIVE=1 Tool[3]:GUN C2 Base[3]:Atego/Axor;%{PE}%R 8.2.2,%MKUKATPSPOT,%CSPOT,%VLIN,%P 1:LIN, 2:SWP_60_7487, 3:, 5:2, 7:L_OLP31, 10:2, 12:#FIRST, 14:#CLO, 16:185, 18:1, 20:0, 22:0, 24:1, 25:NORMAL
$BWDSTART=FALSE
LDAT_ACT=LL_OLP31
FDAT_ACT=FSWP_60_7487
BAS(#CP_PARAMS,LL_OLP31.VEL)
S_ACT.GUN=2
S_ACT.PAIR=SDEFAULT.PAIR
S_ACT.RETR=#CLO
S_ACT.CLO_TM=1
S_ACT.PGNO1=185
S_ACT.PGNO2=SDEFAULT.PGNO2
S_ACT.PRESS1=SDEFAULT.PRESS1
S_ACT.PRESS2=SDEFAULT.PRESS2
S_READY=FALSE
LIN XSWP_60_7487
USERSPOT(#SPOT, S_ACT)
WAIT FOR S_READY
;ENDFOLD

;FOLD ; SWP_60_7489;%{PE}%R 4.1.16,%MKUKATPBASIS,%CCOMMENT,%VNORMAL,%P 2:SWP_60_7489
;ENDFOLD
;FOLD LIN SWP_60_7489 L_OLP32 SPOT Gun=2 RETR CLS PgNo1=185 ACTIVE=1 Tool[3]:GUN C2 Base[3]:Atego/Axor;%{PE}%R 8.2.2,%MKUKATPSPOT,%CSPOT,%VLIN,%P 1:LIN, 2:SWP_60_7489, 3:, 5:2, 7:L_OLP32, 10:2, 12:#FIRST, 14:#CLO, 16:185, 18:1, 20:0, 22:0, 24:1, 25:NORMAL
$BWDSTART=FALSE
LDAT_ACT=LL_OLP32
FDAT_ACT=FSWP_60_7489
BAS(#CP_PARAMS,LL_OLP32.VEL)
S_ACT.GUN=2
S_ACT.PAIR=SDEFAULT.PAIR
S_ACT.RETR=#CLO
S_ACT.CLO_TM=1
S_ACT.PGNO1=185
S_ACT.PGNO2=SDEFAULT.PGNO2
S_ACT.PRESS1=SDEFAULT.PRESS1
S_ACT.PRESS2=SDEFAULT.PRESS2
S_READY=FALSE
LIN XSWP_60_7489
USERSPOT(#SPOT, S_ACT)
WAIT FOR S_READY
;ENDFOLD

;FOLD ; SWP_60_7491;%{PE}%R 4.1.16,%MKUKATPBASIS,%CCOMMENT,%VNORMAL,%P 2:SWP_60_7491
;ENDFOLD
;FOLD LIN SWP_60_7491 L_OLP33 SPOT Gun=2 RETR OPN PgNo1=185 ACTIVE=1 Tool[3]:GUN C2 Base[3]:Atego/Axor;%{PE}%R 8.2.2,%MKUKATPSPOT,%CSPOT,%VLIN,%P 1:LIN, 2:SWP_60_7491, 3:, 5:2, 7:L_OLP33, 10:2, 12:#FIRST, 14:#OPN, 16:185, 18:1, 20:0, 22:0, 24:1, 25:NORMAL
$BWDSTART=FALSE
LDAT_ACT=LL_OLP33
FDAT_ACT=FSWP_60_7491
BAS(#CP_PARAMS,LL_OLP33.VEL)
S_ACT.GUN=2
S_ACT.PAIR=SDEFAULT.PAIR
S_ACT.RETR=#OPN
S_ACT.CLO_TM=1
S_ACT.PGNO1=185
S_ACT.PGNO2=SDEFAULT.PGNO2
S_ACT.PRESS1=SDEFAULT.PRESS1
S_ACT.PRESS2=SDEFAULT.PRESS2
S_READY=FALSE
LIN XSWP_60_7491
USERSPOT(#SPOT, S_ACT)
WAIT FOR S_READY
;ENDFOLD

;FOLD LIN l105  Vel=2.00 m/s L_OLP34 Tool[3]:Gun C02 Base[3]:Atego/Axor;%{PE}%R8.2.19,%MKUKATPBASIS,%CMOVE,%VLIN,%P 1:LIN, 2:l105, 3: , 5:2.00, 7:L_OLP34
$BWDSTART = FALSE
LDAT_ACT= LL_OLP34
FDAT_ACT= Fl105
BAS(#CP_PARAMS,2.00)
LIN Xl105
;ENDFOLD
;FOLD LIN l110  Vel=2.00 m/s L_OLP35 Tool[3]:Gun C02 Base[3]:Atego/Axor;%{PE}%R8.2.19,%MKUKATPBASIS,%CMOVE,%VLIN,%P 1:LIN, 2:l110, 3: , 5:2.00, 7:L_OLP35
$BWDSTART = FALSE
LDAT_ACT= LL_OLP35
FDAT_ACT= Fl110
BAS(#CP_PARAMS,2.00)
LIN Xl110
;ENDFOLD

;FOLD ; SWP_60_7495;%{PE}%R 4.1.16,%MKUKATPBASIS,%CCOMMENT,%VNORMAL,%P 2:SWP_60_7495
;ENDFOLD
;FOLD LIN SWP_60_7495 L_OLP36 SPOT Gun=2 RETR CLS PgNo1=185 ACTIVE=1 Tool[3]:GUN C2 Base[3]:Atego/Axor;%{PE}%R 8.2.2,%MKUKATPSPOT,%CSPOT,%VLIN,%P 1:LIN, 2:SWP_60_7495, 3:, 5:2, 7:L_OLP36, 10:2, 12:#FIRST, 14:#CLO, 16:185, 18:1, 20:0, 22:0, 24:1, 25:NORMAL
$BWDSTART=FALSE
LDAT_ACT=LL_OLP36
FDAT_ACT=FSWP_60_7495
BAS(#CP_PARAMS,LL_OLP36.VEL)
S_ACT.GUN=2
S_ACT.PAIR=SDEFAULT.PAIR
S_ACT.RETR=#CLO
S_ACT.CLO_TM=1
S_ACT.PGNO1=185
S_ACT.PGNO2=SDEFAULT.PGNO2
S_ACT.PRESS1=SDEFAULT.PRESS1
S_ACT.PRESS2=SDEFAULT.PRESS2
S_READY=FALSE
LIN XSWP_60_7495
USERSPOT(#SPOT, S_ACT)
WAIT FOR S_READY
;ENDFOLD

;FOLD ; SWP_60_7497;%{PE}%R 4.1.16,%MKUKATPBASIS,%CCOMMENT,%VNORMAL,%P 2:SWP_60_7497
;ENDFOLD
;FOLD LIN SWP_60_7497 L_OLP37 SPOT Gun=2 RETR CLS PgNo1=185 ACTIVE=1 Tool[3]:GUN C2 Base[3]:Atego/Axor;%{PE}%R 8.2.2,%MKUKATPSPOT,%CSPOT,%VLIN,%P 1:LIN, 2:SWP_60_7497, 3:, 5:2, 7:L_OLP37, 10:2, 12:#FIRST, 14:#CLO, 16:185, 18:1, 20:0, 22:0, 24:1, 25:NORMAL
$BWDSTART=FALSE
LDAT_ACT=LL_OLP37
FDAT_ACT=FSWP_60_7497
BAS(#CP_PARAMS,LL_OLP37.VEL)
S_ACT.GUN=2
S_ACT.PAIR=SDEFAULT.PAIR
S_ACT.RETR=#CLO
S_ACT.CLO_TM=1
S_ACT.PGNO1=185
S_ACT.PGNO2=SDEFAULT.PGNO2
S_ACT.PRESS1=SDEFAULT.PRESS1
S_ACT.PRESS2=SDEFAULT.PRESS2
S_READY=FALSE
LIN XSWP_60_7497
USERSPOT(#SPOT, S_ACT)
WAIT FOR S_READY
;ENDFOLD

;FOLD ; SWP_60_7499;%{PE}%R 4.1.16,%MKUKATPBASIS,%CCOMMENT,%VNORMAL,%P 2:SWP_60_7499
;ENDFOLD
;FOLD LIN SWP_60_7499 L_OLP38 SPOT Gun=2 RETR OPN PgNo1=185 ACTIVE=1 Tool[3]:GUN C2 Base[3]:Atego/Axor;%{PE}%R 8.2.2,%MKUKATPSPOT,%CSPOT,%VLIN,%P 1:LIN, 2:SWP_60_7499, 3:, 5:2, 7:L_OLP38, 10:2, 12:#FIRST, 14:#OPN, 16:185, 18:1, 20:0, 22:0, 24:1, 25:NORMAL
$BWDSTART=FALSE
LDAT_ACT=LL_OLP38
FDAT_ACT=FSWP_60_7499
BAS(#CP_PARAMS,LL_OLP38.VEL)
S_ACT.GUN=2
S_ACT.PAIR=SDEFAULT.PAIR
S_ACT.RETR=#OPN
S_ACT.CLO_TM=1
S_ACT.PGNO1=185
S_ACT.PGNO2=SDEFAULT.PGNO2
S_ACT.PRESS1=SDEFAULT.PRESS1
S_ACT.PRESS2=SDEFAULT.PRESS2
S_READY=FALSE
LIN XSWP_60_7499
USERSPOT(#SPOT, S_ACT)
WAIT FOR S_READY
;ENDFOLD

;FOLD LIN l115 CONT Vel=2 m/s L_OLP39 Tool[3]:GUN C2 Base[3]:Atego/Axor;%{PE}%R 8.2.20,%MKUKATPBASIS,%CMOVE,%VLIN,%P 1:LIN, 2:l115, 3:C_DIS C_DIS, 5:2, 7:L_OLP39
$BWDSTART=FALSE
LDAT_ACT=LL_OLP39
FDAT_ACT=Fl115
BAS(#CP_PARAMS,2)
LIN Xl115 C_DIS C_DIS
;ENDFOLD
;FOLD LIN l120 CONT Vel=2 m/s L_OLP40 Tool[3]:GUN C2 Base[3]:Atego/Axor;%{PE}%R 8.2.20,%MKUKATPBASIS,%CMOVE,%VLIN,%P 1:LIN, 2:l120, 3:C_DIS C_DIS, 5:2, 7:L_OLP40
$BWDSTART=FALSE
LDAT_ACT=LL_OLP40
FDAT_ACT=Fl120
BAS(#CP_PARAMS,2)
LIN Xl120 C_DIS C_DIS
;ENDFOLD
;FOLD LIN l125 CONT Vel=2 m/s CPDAT23 Tool[3]:GUN C2 Base[3]:Atego/Axor;%{PE}%R 8.2.20,%MKUKATPBASIS,%CMOVE,%VLIN,%P 1:LIN, 2:l125, 3:C_DIS C_DIS, 5:2, 7:CPDAT23
$BWDSTART=FALSE
LDAT_ACT=LCPDAT23
FDAT_ACT=Fl125
BAS(#CP_PARAMS,2)
LIN Xl125 C_DIS C_DIS
;ENDFOLD
;FOLD PTP P18 CONT Vel=100 % PDAT13 Tool[3]:GUN C2 Base[3]:Atego/Axor;%{PE}%R 8.2.20,%MKUKATPBASIS,%CMOVE,%VPTP,%P 1:PTP, 2:P18, 3:C_DIS, 5:100, 7:PDAT13
$BWDSTART=FALSE
PDAT_ACT=PPDAT13
FDAT_ACT=FP18
BAS(#PTP_PARAMS,100)
PTP XP18 C_DIS
;ENDFOLD
;FOLD PTP P13 Vel=100 % PDAT10 Tool[3]:GUN C2 Base[3]:Atego/Axor;%{PE}%R 8.2.20,%MKUKATPBASIS,%CMOVE,%VPTP,%P 1:PTP, 2:P13, 3:, 5:100, 7:PDAT10
$BWDSTART=FALSE
PDAT_ACT=PPDAT10
FDAT_ACT=FP13
BAS(#PTP_PARAMS,100)
PTP XP13
;ENDFOLD

IF (NOT(GHOST())) THEN
IF FraesAnf(3) THEN
  f_Fraes_3 ()
ENDIF
ENDIF

END

--- ps_a_stb_res_c02.dat ---
&ACCESS RVO1
&REL 230
&COMMENT Solda Atego STB
&PARAM DISKPATH = KRC:\R1\Program\OLP
DEFDAT  ps_a_stb_res_c02
;FOLD EXTERNAL DECLARATIONS;%{PE}%MKUKATPBASIS,%CEXT,%VCOMMON,%P
;FOLD GRIPPERTECH EXT
EXT  H50 (INT  :IN,INT  :IN,INT  :IN,GRP_TYP  :IN )
;ENDFOLD (GRIPPERTECH EXT)
;FOLD SPOTTECH EXT
EXT  USERSPOT (S_COMMAND  :IN,SPOT_TYPE  :IN )
;ENDFOLD (SPOTTECH EXT)
;FOLD BASISTECH EXT;%{PE}%MKUKATPBASIS,%CEXT,%VEXT,%P
EXT  BAS (BAS_COMMAND  :IN,REAL  :IN )
DECL INT SUCCESS
;ENDFOLD (BASISTECH EXT)
;FOLD USER EXT;%{E}%MKUKATPUSER,%CEXT,%VEXT,%P
;Make your modifications here

;ENDFOLD (USER EXT)
;ENDFOLD (EXTERNAL DECLARATIONS)
DECL FDAT Fl015={TOOL_NO 3,BASE_NO 3,IPO_FRAME #BASE,POINT2[] " "}
DECL E6POS Xl015={X 34.2892494,Y -644.046082,Z 761.163513,A -123.997002,B 73.4720612,C -126.848701,S 18,T 35,E1 0.0,E2 0.0,E3 0.0,E4 0.0,E5 0.0,E6 0.0}
DECL LDAT LL_OLP3={VEL 2.0,ACC 100.0,APO_DIST 0.0,APO_FAC 0.0,ORI_TYP #VAR,CIRC_TYP #BASE,JERK_FAC 50.0}
DECL FDAT Fl030={TOOL_NO 3,BASE_NO 3,IPO_FRAME #BASE,POINT2[] " "}
DECL E6POS Xl030={X 274.340912,Y -703.442017,Z 641.453125,A -54.7125397,B 69.4866562,C -51.1110687,S 18,T 35,E1 0.0,E2 0.0,E3 0.0,E4 0.0,E5 0.0,E6 0.0}
DECL LDAT LL_OLP6={VEL 2.0,ACC 100.0,APO_DIST 30.0,APO_FAC 0.0,ORI_TYP #VAR,CIRC_TYP #BASE,JERK_FAC 50.0}
DECL FDAT Fl035={TOOL_NO 3,BASE_NO 3,IPO_FRAME #BASE,POINT2[] " "}
DECL E6POS Xl035={X 587.583008,Y -653.065002,Z 418.535004,A -24.4300995,B 45.0119019,C -12.2528,S 2,T 35}
DECL LDAT LL_OLP7={VEL 2.0,ACC 100.0,APO_DIST 30.0,APO_FAC 0.0,ORI_TYP #VAR,CIRC_TYP #BASE,JERK_FAC 50.0}
DECL FDAT Fl040={TOOL_NO 3,BASE_NO 3,IPO_FRAME #BASE,POINT2[] " "}
DECL E6POS Xl040={X 713.926392,Y -668.47052,Z 338.3591,A -21.6110992,B 32.5932884,C -7.47571993,S 18,T 35,E1 0.0,E2 0.0,E3 0.0,E4 0.0,E5 0.0,E6 0.0}
DECL LDAT LL_OLP8={VEL 2.0,ACC 100.0,APO_DIST 150.0,APO_FAC 0.0,ORI_TYP #VAR,CIRC_TYP #BASE,JERK_FAC 50.0}
DECL FDAT Fl045={TOOL_NO 3,BASE_NO 3,IPO_FRAME #BASE,POINT2[] " "}
DECL E6POS Xl045={X 765.193115,Y -1115.46997,Z 133.110596,A -16.9657192,B 14.9491901,C -20.2578106,S 18,T 3,E1 0.0,E2 0.0,E3 0.0,E4 0.0,E5 0.0,E6 0.0}
DECL LDAT LL_OLP9={VEL 2.0,ACC 100.0,APO_DIST 150.0,APO_FAC 0.0,ORI_TYP #VAR,CIRC_TYP #BASE,JERK_FAC 50.0}
DECL FDAT Fl050={TOOL_NO 3,BASE_NO 3,IPO_FRAME #BASE,POINT2[] " "}
DECL E6POS Xl050={X 746.955017,Y -2151.34399,Z 121.584,A -16.3197002,B 12.0216999,C -22.6774998,S 2,T 3}
DECL FDAT Fl060={TOOL_NO 3,BASE_NO 3,IPO_FRAME #BASE,POINT2[] " "}
DECL PDAT PP_OLP2={VEL 100.0,ACC 100.0,APO_DIST 100.0,APO_MODE #CDIS}
DECL E6POS Xl060={X 1158.77795,Y -1627.54797,Z 929.039001,A 43.2759018,B -40.0696983,C 26.0069008,S 6,T 19}
DECL FDAT Fl065={TOOL_NO 3,BASE_NO 3,IPO_FRAME #BASE,POINT2[] " "}
DECL PDAT PP_OLP3={VEL 100.0,ACC 100.0,APO_DIST 30.0,APO_MODE #CDIS}
DECL E6POS Xl065={X 868.09668,Y -1244.59497,Z 1101.58606,A 29.2385902,B -63.5374794,C 57.4689713,S 22,T 19,E1 0.0,E2 0.0,E3 0.0,E4 0.0,E5 0.0,E6 0.0}
DECL FDAT Fl070={TOOL_NO 3,BASE_NO 3,IPO_FRAME #BASE,POINT2[] " "}
DECL PDAT PP_OLP4={VEL 100.0,ACC 100.0,APO_DIST 30.0,APO_MODE #CDIS}
DECL E6POS Xl070={X 814.102905,Y -929.709717,Z 1165.05896,A 29.5652695,B -64.2360001,C 60.087719,S 22,T 19,E1 0.0,E2 0.0,E3 0.0,E4 0.0,E5 0.0,E6 0.0}
DECL E6POS XSWP_60_7787={X 556.090027,Y -970.939697,Z 1302.49805,A 143.935699,B -83.3155518,C -51.7020683,S 22,T 19,E1 0.0,E2 0.0,E3 0.0,E4 0.0,E5 0.0,E6 0.0}
DECL FDAT FSWP_60_7787={TOOL_NO 3,BASE_NO 3,IPO_FRAME #BASE,POINT2[] " "}
DECL LDAT LL_OLP12={VEL 2.0,ACC 100.0,APO_DIST 0.0,APO_FAC 0.0,ORI_TYP #VAR,CIRC_TYP #BASE,JERK_FAC 50.0}
DECL E6POS XSWP_60_7789={X 584.018677,Y -975.191223,Z 1304.28101,A 144.007706,B -83.3220673,C -54.6376801,S 18,T 43,E1 0.0,E2 0.0,E3 0.0,E4 0.0,E5 0.0,E6 0.0}
DECL FDAT FSWP_60_7789={TOOL_NO 3,BASE_NO 3,IPO_FRAME #BASE,POINT2[] " "}
DECL LDAT LL_OLP13={VEL 2.0,ACC 100.0,APO_DIST 0.0,APO_FAC 0.0,ORI_TYP #VAR,CIRC_TYP #BASE,JERK_FAC 50.0}
DECL E6POS XSWP_60_7791={X 613.497314,Y -974.923523,Z 1306.802,A 144.014694,B -83.3241119,C -54.6452789,S 18,T 43,E1 0.0,E2 0.0,E3 0.0,E4 0.0,E5 0.0,E6 0.0}
DECL FDAT FSWP_60_7791={TOOL_NO 3,BASE_NO 3,IPO_FRAME #BASE,POINT2[] " "}
DECL LDAT LL_OLP14={VEL 2.0,ACC 100.0,APO_DIST 0.0,APO_FAC 0.0,ORI_TYP #VAR,CIRC_TYP #BASE,JERK_FAC 50.0}
DECL E6POS XSWP_60_7795={X 702.547974,Y -976.360229,Z 1310.90698,A 26.1141891,B -81.5289536,C 62.8172913,S 22,T 19,E1 0.0,E2 0.0,E3 0.0,E4 0.0,E5 0.0,E6 0.0}
DECL FDAT FSWP_60_7795={TOOL_NO 3,BASE_NO 3,IPO_FRAME #BASE,POINT2[] " "}
DECL LDAT LL_OLP16={VEL 2.0,ACC 100.0,APO_DIST 0.0,APO_FAC 0.0,ORI_TYP #VAR,CIRC_TYP #BASE,JERK_FAC 50.0}
DECL E6POS XSWP_60_7797={X 744.221313,Y -976.517883,Z 1312.43994,A 26.1132603,B -81.5287933,C 62.8183212,S 22,T 19,E1 0.0,E2 0.0,E3 0.0,E4 0.0,E5 0.0,E6 0.0}
DECL FDAT FSWP_60_7797={TOOL_NO 3,BASE_NO 3,IPO_FRAME #BASE,POINT2[] " "}
DECL LDAT LL_OLP17={VEL 2.0,ACC 100.0,APO_DIST 0.0,APO_FAC 0.0,ORI_TYP #VAR,CIRC_TYP #BASE,JERK_FAC 50.0}
DECL E6POS XSWP_60_7799={X 790.635193,Y -976.77002,Z 1313.89795,A 26.1131706,B -81.5296173,C 62.8176003,S 22,T 19,E1 0.0,E2 0.0,E3 0.0,E4 0.0,E5 0.0,E6 0.0}
DECL FDAT FSWP_60_7799={TOOL_NO 3,BASE_NO 3,IPO_FRAME #BASE,POINT2[] " "}
DECL LDAT LL_OLP18={VEL 2.0,ACC 100.0,APO_DIST 0.0,APO_FAC 0.0,ORI_TYP #VAR,CIRC_TYP #BASE,JERK_FAC 50.0}
DECL E6POS XSWP_60_7801={X 838.134583,Y -978.93042,Z 1314.93604,A 26.1214104,B -81.5290985,C 62.8091202,S 22,T 19,E1 0.0,E2 0.0,E3 0.0,E4 0.0,E5 0.0,E6 0.0}
DECL FDAT FSWP_60_7801={TOOL_NO 3,BASE_NO 3,IPO_FRAME #BASE,POINT2[] " "}
DECL LDAT LL_OLP19={VEL 2.0,ACC 100.0,APO_DIST 0.0,APO_FAC 0.0,ORI_TYP #VAR,CIRC_TYP #BASE,JERK_FAC 50.0}
DECL E6POS XSWP_60_7803={X 879.105103,Y -979.47998,Z 1316.29504,A 26.1255798,B -81.5288086,C 62.8046112,S 22,T 19,E1 0.0,E2 0.0,E3 0.0,E4 0.0,E5 0.0,E6 0.0}
DECL FDAT FSWP_60_7803={TOOL_NO 3,BASE_NO 3,IPO_FRAME #BASE,POINT2[] " "}
DECL LDAT LL_OLP20={VEL 2.0,ACC 100.0,APO_DIST 0.0,APO_FAC 0.0,ORI_TYP #VAR,CIRC_TYP #BASE,JERK_FAC 50.0}
DECL E6POS XSWP_60_7807={X 972.604675,Y -980.853088,Z 1320.021,A 26.1273499,B -81.5320511,C 62.8050995,S 22,T 19,E1 0.0,E2 0.0,E3 0.0,E4 0.0,E5 0.0,E6 0.0}
DECL FDAT FSWP_60_7807={TOOL_NO 3,BASE_NO 3,IPO_FRAME #BASE,POINT2[] " "}
DECL LDAT LL_OLP21={VEL 2.0,ACC 100.0,APO_DIST 0.0,APO_FAC 0.0,ORI_TYP #VAR,CIRC_TYP #BASE,JERK_FAC 50.0}
DECL E6POS XSWP_60_7809={X 1020.008,Y -981.762024,Z 1320.86694,A 26.1021709,B -81.5283127,C 62.8302803,S 18,T 43,E1 0.0,E2 0.0,E3 0.0,E4 0.0,E5 0.0,E6 0.0}
DECL FDAT FSWP_60_7809={TOOL_NO 3,BASE_NO 3,IPO_FRAME #BASE,POINT2[] " "}
DECL LDAT LL_OLP22={VEL 2.0,ACC 100.0,APO_DIST 0.0,APO_FAC 0.0,ORI_TYP #VAR,CIRC_TYP #BASE,JERK_FAC 50.0}
DECL E6POS XSWP_60_7811={X 1062.04297,Y -981.887817,Z 1321.88403,A 26.1206608,B -81.5300064,C 62.8098907,S 22,T 19,E1 0.0,E2 0.0,E3 0.0,E4 0.0,E5 0.0,E6 0.0}
DECL FDAT FSWP_60_7811={TOOL_NO 3,BASE_NO 3,IPO_FRAME #BASE,POINT2[] " "}
DECL LDAT LL_OLP23={VEL 2.0,ACC 100.0,APO_DIST 0.0,APO_FAC 0.0,ORI_TYP #VAR,CIRC_TYP #BASE,JERK_FAC 50.0}
DECL E6POS XSWP_60_7813={X 1102.54004,Y -982.899414,Z 1323.276,A 26.1103706,B -81.5286636,C 62.8202515,S 22,T 19,E1 0.0,E2 0.0,E3 0.0,E4 0.0,E5 0.0,E6 0.0}
DECL FDAT FSWP_60_7813={TOOL_NO 3,BASE_NO 3,IPO_FRAME #BASE,POINT2[] " "}
DECL LDAT LL_OLP24={VEL 2.0,ACC 100.0,APO_DIST 0.0,APO_FAC 0.0,ORI_TYP #VAR,CIRC_TYP #BASE,JERK_FAC 50.0}
DECL E6POS XSWP_60_7815={X 1147.95996,Y -980.301575,Z 1324.172,A 26.1117191,B -81.5287018,C 62.8188019,S 22,T 19,E1 0.0,E2 0.0,E3 0.0,E4 0.0,E5 0.0,E6 0.0}
DECL FDAT FSWP_60_7815={TOOL_NO 3,BASE_NO 3,IPO_FRAME #BASE,POINT2[] " "}
DECL LDAT LL_OLP25={VEL 2.0,ACC 100.0,APO_DIST 0.0,APO_FAC 0.0,ORI_TYP #VAR,CIRC_TYP #BASE,JERK_FAC 50.0}
DECL FDAT Fl085={TOOL_NO 3,BASE_NO 3,IPO_FRAME #BASE,POINT2[] " "}
DECL E6POS Xl085={X 1164.30798,Y -948.935486,Z 1258.81995,A 17.7583904,B -81.8330536,C 71.0863037,S 22,T 19,E1 0.0,E2 0.0,E3 0.0,E4 0.0,E5 0.0,E6 0.0}
DECL LDAT LL_OLP27={VEL 2.0,ACC 100.0,APO_DIST 150.0,APO_FAC 0.0,ORI_TYP #VAR,CIRC_TYP #BASE,JERK_FAC 50.0}
DECL FDAT Fl090={TOOL_NO 3,BASE_NO 3,IPO_FRAME #BASE,POINT2[] " "}
DECL E6POS Xl090={X 983.369995,Y -1478.85596,Z 590.278015,A 179.957108,B -45.9999008,C -90.0,S 6,T 19}
DECL LDAT LL_OLP28={VEL 2.0,ACC 100.0,APO_DIST 150.0,APO_FAC 0.0,ORI_TYP #VAR,CIRC_TYP #BASE,JERK_FAC 50.0}
DECL FDAT Fl095={TOOL_NO 3,BASE_NO 3,IPO_FRAME #BASE,POINT2[] " "}
DECL E6POS Xl095={X 1322.44702,Y -1291.22498,Z 42.4953308,A 179.958099,B -15.9995604,C -90.0038834,S 22,T 19,E1 0.0,E2 0.0,E3 0.0,E4 0.0,E5 0.0,E6 0.0}
DECL LDAT LL_OLP29={VEL 2.0,ACC 100.0,APO_DIST 30.0,APO_FAC 0.0,ORI_TYP #VAR,CIRC_TYP #BASE,JERK_FAC 50.0}
DECL FDAT Fl100={TOOL_NO 3,BASE_NO 3,IPO_FRAME #BASE,POINT2[] " "}
DECL E6POS Xl100={X 1301.61499,Y -1007.51001,Z 77.1176071,A 179.957001,B -16.00037,C -89.9989929,S 22,T 19,E1 0.0,E2 0.0,E3 0.0,E4 0.0,E5 0.0,E6 0.0}
DECL LDAT LL_OLP30={VEL 2.0,ACC 100.0,APO_DIST 0.0,APO_FAC 0.0,ORI_TYP #VAR,CIRC_TYP #BASE,JERK_FAC 50.0}
DECL FDAT FSWP_60_7487={TOOL_NO 3,BASE_NO 3,IPO_FRAME #BASE,POINT2[] " "}
DECL E6POS XSWP_60_7487={X 1306.44397,Y -1021.547,Z 118.262802,A 179.322403,B -25.28022,C -90.9719391,S 18,T 43,E1 0.0,E2 0.0,E3 0.0,E4 0.0,E5 0.0,E6 0.0}
DECL LDAT LL_OLP31={VEL 2.0,ACC 100.0,APO_DIST 0.0,APO_FAC 0.0,ORI_TYP #VAR,CIRC_TYP #BASE,JERK_FAC 50.0}
DECL FDAT FSWP_60_7489={TOOL_NO 3,BASE_NO 3,IPO_FRAME #BASE,POINT2[] " "}
DECL E6POS XSWP_60_7489={X 1339.98206,Y -1023.56598,Z 120.081001,A 179.952698,B -20.9994793,C -93.3431702,S 18,T 43,E1 0.0,E2 0.0,E3 0.0,E4 0.0,E5 0.0,E6 0.0}
DECL LDAT LL_OLP32={VEL 2.0,ACC 100.0,APO_DIST 0.0,APO_FAC 0.0,ORI_TYP #VAR,CIRC_TYP #BASE,JERK_FAC 50.0}
DECL FDAT FSWP_60_7491={TOOL_NO 3,BASE_NO 3,IPO_FRAME #BASE,POINT2[] " "}
DECL E6POS XSWP_60_7491={X 1370.55298,Y -1021.91803,Z 121.484901,A -179.790604,B -20.8528404,C -93.2146988,S 18,T 43,E1 0.0,E2 0.0,E3 0.0,E4 0.0,E5 0.0,E6 0.0}
DECL LDAT LL_OLP33={VEL 2.0,ACC 100.0,APO_DIST 0.0,APO_FAC 0.0,ORI_TYP #VAR,CIRC_TYP #BASE,JERK_FAC 50.0}
DECL FDAT Fl105={TOOL_NO 3,BASE_NO 3,IPO_FRAME #BASE,POINT2[] " "}
DECL E6POS Xl105={X 1373.94495,Y -1013.10602,Z 88.1965637,A 179.956894,B -18.0000401,C -89.9994507,S 22,T 19,E1 0.0,E2 0.0,E3 0.0,E4 0.0,E5 0.0,E6 0.0}
DECL LDAT LL_OLP34={VEL 2.0,ACC 100.0,APO_DIST 0.0,APO_FAC 0.0,ORI_TYP #VAR,CIRC_TYP #BASE,JERK_FAC 50.0}
DECL FDAT Fl110={TOOL_NO 3,BASE_NO 3,IPO_FRAME #BASE,POINT2[] " "}
DECL E6POS Xl110={X 1469.69604,Y -999.753174,Z 86.6159668,A 179.956894,B -19.0000801,C -89.9993668,S 22,T 19,E1 0.0,E2 0.0,E3 0.0,E4 0.0,E5 0.0,E6 0.0}
DECL LDAT LL_OLP35={VEL 2.0,ACC 100.0,APO_DIST 0.0,APO_FAC 0.0,ORI_TYP #VAR,CIRC_TYP #BASE,JERK_FAC 50.0}
DECL FDAT FSWP_60_7495={TOOL_NO 3,BASE_NO 3,IPO_FRAME #BASE,POINT2[] " "}
DECL E6POS XSWP_60_7495={X 1442.27197,Y -1019.48102,Z 122.377296,A 179.957199,B -20.9995899,C -93.1918564,S 22,T 19,E1 0.0,E2 0.0,E3 0.0,E4 0.0,E5 0.0,E6 0.0}
DECL LDAT LL_OLP36={VEL 2.0,ACC 100.0,APO_DIST 0.0,APO_FAC 0.0,ORI_TYP #VAR,CIRC_TYP #BASE,JERK_FAC 50.0}
DECL FDAT FSWP_60_7497={TOOL_NO 3,BASE_NO 3,IPO_FRAME #BASE,POINT2[] " "}
DECL E6POS XSWP_60_7497={X 1479.71106,Y -1018.96399,Z 124.096703,A -179.6689,B -20.9927502,C -93.8000717,S 18,T 43,E1 0.0,E2 0.0,E3 0.0,E4 0.0,E5 0.0,E6 0.0}
DECL LDAT LL_OLP37={VEL 2.0,ACC 100.0,APO_DIST 0.0,APO_FAC 0.0,ORI_TYP #VAR,CIRC_TYP #BASE,JERK_FAC 50.0}
DECL FDAT FSWP_60_7499={TOOL_NO 3,BASE_NO 3,IPO_FRAME #BASE,POINT2[] " "}
DECL E6POS XSWP_60_7499={X 1519.71802,Y -1018.96802,Z 124.852798,A -179.660904,B -20.9865093,C -93.8057938,S 18,T 43,E1 0.0,E2 0.0,E3 0.0,E4 0.0,E5 0.0,E6 0.0}
DECL LDAT LL_OLP38={VEL 2.0,ACC 100.0,APO_DIST 0.0,APO_FAC 0.0,ORI_TYP #VAR,CIRC_TYP #BASE,JERK_FAC 50.0}
DECL FDAT Fl115={TOOL_NO 3,BASE_NO 3,IPO_FRAME #BASE,POINT2[] " "}
DECL E6POS Xl115={X 1563.23596,Y -1006.01099,Z 70.940239,A 179.949402,B -20.9986,C -89.9980469,S 22,T 19,E1 0.0,E2 0.0,E3 0.0,E4 0.0,E5 0.0,E6 0.0}
DECL LDAT LL_OLP39={VEL 2.0,ACC 100.0,APO_DIST 150.0,APO_FAC 0.0,ORI_TYP #VAR,CIRC_TYP #BASE,JERK_FAC 50.0}
DECL FDAT Fl120={TOOL_NO 3,BASE_NO 3,IPO_FRAME #BASE,POINT2[] " "}
DECL E6POS Xl120={X 1563.09998,Y -1231.07898,Z 75.473999,A 179.957108,B -20.9999008,C -90.0,S 6,T 19}
DECL LDAT LL_OLP40={VEL 2.0,ACC 100.0,APO_DIST 150.0,APO_FAC 0.0,ORI_TYP #VAR,CIRC_TYP #BASE,JERK_FAC 50.0}
DECL FDAT Fl125={TOOL_NO 3,BASE_NO 3,IPO_FRAME #BASE,POINT2[] " "}
DECL E6POS Xl125={X 1668.59998,Y -1631.57996,Z 177.973999,A 179.957108,B -46.0,C -90.0,S 6,T 19}
DECL BASIS_SUGG_T LAST_BASIS={POINT1[] "P18                     ",POINT2[] "P18                     ",CP_PARAMS[] "CPDAT19                 ",PTP_PARAMS[] "PDAT13                  ",CONT[] "                        ",CP_VEL[] "2                       ",PTP_VEL[] "100                     ",SYNC_PARAMS[] "SYNCDAT                 ",SPL_NAME[] "S0                      "}
DECL PDAT PP_OLP6={VEL 100.0,ACC 100.0,APO_DIST 0.0}
DECL E6POS Xl006={X 746.955017,Y -2151.34399,Z 121.584,A -16.3197002,B 12.0216999,C -22.6774998,S 2,T 3}
DECL FDAT Fl006={TOOL_NO 3,BASE_NO 3,IPO_FRAME #BASE,POINT2[] " "}
DECL LDAT LL_OLP42={VEL 2.0,ACC 100.0,APO_DIST 30.0,APO_FAC 0.0,ORI_TYP #VAR,CIRC_TYP #BASE,JERK_FAC 50.0}
DECL E6POS Xl011={X 745.054077,Y -1210.42102,Z 45.7849503,A -16.3183804,B 12.0204601,C -22.6786194,S 18,T 3,E1 0.0,E2 0.0,E3 0.0,E4 0.0,E5 0.0,E6 0.0}
DECL FDAT Fl011={TOOL_NO 3,BASE_NO 3,IPO_FRAME #BASE,POINT2[] " "}
DECL E6POS Xl016={X 960.239685,Y -695.417419,Z 224.849792,A -18.2002106,B 11.2452402,C -1.07748699,S 18,T 3,E1 0.0,E2 0.0,E3 0.0,E4 0.0,E5 0.0,E6 0.0}
DECL FDAT Fl016={TOOL_NO 3,BASE_NO 3,IPO_FRAME #BASE,POINT2[] " "}
DECL LDAT LL_OLP44={VEL 2.0,ACC 100.0,APO_DIST 10.0,APO_FAC 0.0,ORI_TYP #VAR,CIRC_TYP #BASE,JERK_FAC 50.0}
DECL E6POS Xl021={X 587.583008,Y -653.065002,Z 418.535004,A -24.4300995,B 45.0119019,C -12.2528,S 2,T 35}
DECL FDAT Fl021={TOOL_NO 3,BASE_NO 3,IPO_FRAME #BASE,POINT2[] " "}
DECL LDAT LL_OLP45={VEL 2.0,ACC 100.0,APO_DIST 10.0,APO_FAC 0.0,ORI_TYP #VAR,CIRC_TYP #BASE,JERK_FAC 50.0}
DECL E6POS Xl026={X 343.014008,Y -642.028076,Z 721.553772,A -44.0348091,B 69.0998383,C -36.2288399,S 18,T 35,E1 0.0,E2 0.0,E3 0.0,E4 0.0,E5 0.0,E6 0.0}
DECL FDAT Fl026={TOOL_NO 3,BASE_NO 3,IPO_FRAME #BASE,POINT2[] " "}
DECL LDAT LL_OLP46={VEL 2.0,ACC 100.0,APO_DIST 10.0,APO_FAC 0.0,ORI_TYP #VAR,CIRC_TYP #BASE,JERK_FAC 50.0}
DECL E6POS Xl031={X 328.106598,Y -647.627686,Z 744.279175,A -69.6208572,B 74.6609573,C -62.4694595,S 18,T 35,E1 0.0,E2 0.0,E3 0.0,E4 0.0,E5 0.0,E6 0.0}
DECL FDAT Fl031={TOOL_NO 3,BASE_NO 3,IPO_FRAME #BASE,POINT2[] " "}
DECL LDAT LL_OLP47={VEL 2.0,ACC 100.0,APO_DIST 10.0,APO_FAC 0.0,ORI_TYP #VAR,CIRC_TYP #BASE,JERK_FAC 50.0}
DECL E6POS Xl036={X 129.093597,Y -809.958801,Z 712.43811,A -122.0411,B 73.8237534,C -124.462097,S 18,T 35,E1 0.0,E2 0.0,E3 0.0,E4 0.0,E5 0.0,E6 0.0}
DECL FDAT Fl036={TOOL_NO 3,BASE_NO 3,IPO_FRAME #BASE,POINT2[] " "}
DECL LDAT LL_OLP48={VEL 2.0,ACC 100.0,APO_DIST 10.0,APO_FAC 0.0,ORI_TYP #VAR,CIRC_TYP #BASE,JERK_FAC 50.0}
DECL E6POS Xl041={X 111.864998,Y -869.716003,Z 602.434021,A -124.114799,B 73.5134964,C -126.966202,S 2,T 35}
DECL FDAT Fl041={TOOL_NO 3,BASE_NO 3,IPO_FRAME #BASE,POINT2[] " "}
DECL LDAT LL_OLP49={VEL 2.0,ACC 100.0,APO_DIST 0.0,APO_FAC 0.0,ORI_TYP #VAR,CIRC_TYP #BASE,JERK_FAC 50.0}
DECL E6POS XSWP_60_7909={X 133.371994,Y -867.335022,Z 595.832703,A -114.748299,B 75.1414413,C -123.0653,S 18,T 35,E1 0.0,E2 0.0,E3 0.0,E4 0.0,E5 0.0,E6 0.0}
DECL FDAT FSWP_60_7909={TOOL_NO 3,BASE_NO 3,IPO_FRAME #BASE,POINT2[] " "}
DECL E6POS XSWP_60_7907={X 129.194901,Y -831.90509,Z 596.822327,A -114.727898,B 75.1295319,C -117.925201,S 18,T 35,E1 0.0,E2 0.0,E3 0.0,E4 0.0,E5 0.0,E6 0.0}
DECL FDAT FSWP_60_7907={TOOL_NO 3,BASE_NO 3,IPO_FRAME #BASE,POINT2[] " ",TQ_STATE FALSE}
DECL LDAT LL_OLP51={VEL 2.0,ACC 100.0,APO_DIST 0.0,APO_FAC 0.0,ORI_TYP #VAR,CIRC_TYP #BASE,JERK_FAC 50.0}
DECL E6POS XSWP_60_7905={X 118.433098,Y -758.154419,Z 595.061096,A -99.7300873,B 76.5231171,C -103.376701,S 18,T 35,E1 0.0,E2 0.0,E3 0.0,E4 0.0,E5 0.0,E6 0.0}
DECL FDAT FSWP_60_7905={TOOL_NO 3,BASE_NO 3,IPO_FRAME #BASE,POINT2[] " "}
DECL LDAT LL_OLP52={VEL 2.0,ACC 100.0,APO_DIST 0.0,APO_FAC 0.0,ORI_TYP #VAR,CIRC_TYP #BASE,JERK_FAC 50.0}
DECL E6POS XSWP_60_7903={X 114.066704,Y -728.865417,Z 595.601318,A -111.010101,B 80.2996597,C -114.061897,S 18,T 35,E1 0.0,E2 0.0,E3 0.0,E4 0.0,E5 0.0,E6 0.0}
DECL FDAT FSWP_60_7903={TOOL_NO 3,BASE_NO 3,IPO_FRAME #BASE,POINT2[] " "}
DECL LDAT LL_OLP53={VEL 2.0,ACC 100.0,APO_DIST 0.0,APO_FAC 0.0,ORI_TYP #VAR,CIRC_TYP #BASE,JERK_FAC 50.0}
DECL E6POS XSWP_60_7901={X 112.080597,Y -698.418274,Z 594.289795,A -111.004402,B 80.2971268,C -114.0597,S 18,T 35,E1 0.0,E2 0.0,E3 0.0,E4 0.0,E5 0.0,E6 0.0}
DECL FDAT FSWP_60_7901={TOOL_NO 3,BASE_NO 3,IPO_FRAME #BASE,POINT2[] " "}
DECL LDAT LL_OLP54={VEL 2.0,ACC 100.0,APO_DIST 0.0,APO_FAC 0.0,ORI_TYP #VAR,CIRC_TYP #BASE,JERK_FAC 50.0}
DECL E6POS XSWP_60_7329={X 109.463699,Y -668.892273,Z 593.50531,A -111.027702,B 80.2984772,C -114.077797,S 18,T 35,E1 0.0,E2 0.0,E3 0.0,E4 0.0,E5 0.0,E6 0.0}
DECL FDAT FSWP_60_7329={TOOL_NO 3,BASE_NO 3,IPO_FRAME #BASE,POINT2[] " "}
DECL LDAT LL_OLP55={VEL 2.0,ACC 100.0,APO_DIST 0.0,APO_FAC 0.0,ORI_TYP #VAR,CIRC_TYP #BASE,JERK_FAC 50.0}
DECL E6POS XSWP_60_7893={X 102.933197,Y -581.955078,Z 592.471802,A -111.066597,B 80.2849808,C -110.9729,S 18,T 35,E1 0.0,E2 0.0,E3 0.0,E4 0.0,E5 0.0,E6 0.0}
DECL FDAT FSWP_60_7893={TOOL_NO 3,BASE_NO 3,IPO_FRAME #BASE,POINT2[] " "}
DECL LDAT LL_OLP56={VEL 2.0,ACC 100.0,APO_DIST 0.0,APO_FAC 0.0,ORI_TYP #VAR,CIRC_TYP #BASE,JERK_FAC 50.0}
DECL E6POS XSWP_60_7891={X 101.524597,Y -547.288513,Z 593.114197,A -152.9216,B 84.2263412,C -151.278503,S 18,T 35,E1 0.0,E2 0.0,E3 0.0,E4 0.0,E5 0.0,E6 0.0}
DECL FDAT FSWP_60_7891={TOOL_NO 3,BASE_NO 3,IPO_FRAME #BASE,POINT2[] " "}
DECL LDAT LL_OLP57={VEL 2.0,ACC 100.0,APO_DIST 0.0,APO_FAC 0.0,ORI_TYP #VAR,CIRC_TYP #BASE,JERK_FAC 50.0}
DECL E6POS XSWP_60_7889={X 96.6015015,Y -514.959473,Z 593.594604,A -155.411804,B 84.517868,C -154.861099,S 18,T 35,E1 0.0,E2 0.0,E3 0.0,E4 0.0,E5 0.0,E6 0.0}
DECL FDAT FSWP_60_7889={TOOL_NO 3,BASE_NO 3,IPO_FRAME #BASE,POINT2[] " "}
DECL LDAT LL_OLP58={VEL 2.0,ACC 100.0,APO_DIST 0.0,APO_FAC 0.0,ORI_TYP #VAR,CIRC_TYP #BASE,JERK_FAC 50.0}
DECL E6POS XSWP_60_7887={X 94.4030533,Y -481.634491,Z 592.563904,A -106.012802,B 71.1153336,C -109.609703,S 18,T 35,E1 0.0,E2 0.0,E3 0.0,E4 0.0,E5 0.0,E6 0.0}
DECL FDAT FSWP_60_7887={TOOL_NO 3,BASE_NO 3,IPO_FRAME #BASE,POINT2[] " "}
DECL LDAT LL_OLP59={VEL 2.0,ACC 100.0,APO_DIST 0.0,APO_FAC 0.0,ORI_TYP #VAR,CIRC_TYP #BASE,JERK_FAC 50.0}
DECL E6POS XSWP_60_7885={X 97.2438431,Y -448.784912,Z 593.254822,A -109.851997,B 72.9981918,C -112.344902,S 18,T 35,E1 0.0,E2 0.0,E3 0.0,E4 0.0,E5 0.0,E6 0.0}
DECL FDAT FSWP_60_7885={TOOL_NO 3,BASE_NO 3,IPO_FRAME #BASE,POINT2[] " "}
DECL LDAT LL_OLP60={VEL 2.0,ACC 100.0,APO_DIST 0.0,APO_FAC 0.0,ORI_TYP #VAR,CIRC_TYP #BASE,JERK_FAC 50.0}
DECL E6POS XSWP_60_7883={X 95.7695236,Y -416.566406,Z 592.989685,A -113.248596,B 74.3328934,C -114.915298,S 18,T 35,E1 0.0,E2 0.0,E3 0.0,E4 0.0,E5 0.0,E6 0.0}
DECL FDAT FSWP_60_7883={TOOL_NO 3,BASE_NO 3,IPO_FRAME #BASE,POINT2[] " "}
DECL LDAT LL_OLP61={VEL 2.0,ACC 100.0,APO_DIST 0.0,APO_FAC 0.0,ORI_TYP #VAR,CIRC_TYP #BASE,JERK_FAC 50.0}
DECL E6POS XSWP_60_7881={X 93.8571472,Y -383.756012,Z 593.202026,A -121.905296,B 78.0303192,C -124.632698,S 18,T 35,E1 0.0,E2 0.0,E3 0.0,E4 0.0,E5 0.0,E6 0.0}
DECL FDAT FSWP_60_7881={TOOL_NO 3,BASE_NO 3,IPO_FRAME #BASE,POINT2[] " "}
DECL LDAT LCPDAT1={VEL 2.0,ACC 100.0,APO_DIST 100.0,APO_FAC 50.0,AXIS_VEL 100.0,AXIS_ACC 100.0,ORI_TYP #VAR,CIRC_TYP #BASE,JERK_FAC 50.0,GEAR_JERK 50.0,EXAX_IGN 0}
DECL E6POS XP4={X 54.6556282,Y -541.398315,Z 612.695313,A -158.196899,B 83.6885376,C -157.655106,S 18,T 35,E1 0.0,E2 0.0,E3 0.0,E4 0.0,E5 0.0,E6 0.0}
DECL FDAT FP4={TOOL_NO 3,BASE_NO 3,IPO_FRAME #BASE,POINT2[] " ",TQ_STATE FALSE}
DECL LDAT LCPDAT4={VEL 2.0,ACC 100.0,APO_DIST 10.0,APO_FAC 50.0,AXIS_VEL 100.0,AXIS_ACC 100.0,ORI_TYP #VAR,CIRC_TYP #BASE,JERK_FAC 50.0,GEAR_JERK 50.0,EXAX_IGN 0}
DECL E6POS XP5={X 57.6877289,Y -480.831787,Z 603.130127,A -118.843903,B 79.8543396,C -120.822701,S 18,T 35,E1 0.0,E2 0.0,E3 0.0,E4 0.0,E5 0.0,E6 0.0}
DECL FDAT FP5={TOOL_NO 3,BASE_NO 3,IPO_FRAME #BASE,POINT2[] " ",TQ_STATE FALSE}
DECL LDAT LCPDAT5={VEL 2.0,ACC 90.0,APO_DIST 10.0,APO_FAC 50.0,AXIS_VEL 100.0,AXIS_ACC 100.0,ORI_TYP #VAR,CIRC_TYP #BASE,JERK_FAC 50.0,GEAR_JERK 50.0,EXAX_IGN 0}
DECL E6POS XP7={X 684.034424,Y -664.895325,Z 365.229309,A -22.2569199,B 35.8561401,C -8.6238451,S 18,T 35,E1 0.0,E2 0.0,E3 0.0,E4 0.0,E5 0.0,E6 0.0}
DECL FDAT FP7={TOOL_NO 3,BASE_NO 3,IPO_FRAME #BASE,POINT2[] " ",TQ_STATE FALSE}
DECL LDAT LCPDAT7={VEL 2.0,ACC 100.0,APO_DIST 0.0,APO_FAC 50.0,AXIS_VEL 100.0,AXIS_ACC 100.0,ORI_TYP #VAR,CIRC_TYP #BASE,JERK_FAC 50.0,GEAR_JERK 50.0,EXAX_IGN 0}
DECL E6POS XP8={X 687.160217,Y -664.176697,Z 347.525391,A -22.0968399,B 35.009449,C -8.33810997,S 18,T 35,E1 0.0,E2 0.0,E3 0.0,E4 0.0,E5 0.0,E6 0.0}
DECL FDAT FP8={TOOL_NO 3,BASE_NO 3,IPO_FRAME #BASE,POINT2[] " ",TQ_STATE FALSE}
DECL LDAT LCPDAT8={VEL 2.0,ACC 100.0,APO_DIST 10.0,APO_FAC 50.0,AXIS_VEL 100.0,AXIS_ACC 100.0,ORI_TYP #VAR,CIRC_TYP #BASE,JERK_FAC 50.0,GEAR_JERK 50.0,EXAX_IGN 0}
DECL PDAT PPDAT4={VEL 100.0,ACC 100.0,APO_DIST 100.0,GEAR_JERK 50.0}
DECL E6POS XP9={X 621.228516,Y -949.713989,Z 1247.75903,A 77.9962616,B -83.615921,C 13.7808304,S 22,T 19,E1 0.0,E2 0.0,E3 0.0,E4 0.0,E5 0.0,E6 0.0}
DECL FDAT FP9={TOOL_NO 3,BASE_NO 3,IPO_FRAME #BASE,POINT2[] " ",TQ_STATE FALSE}
DECL LDAT LCPDAT9={VEL 2.0,ACC 100.0,APO_DIST 10.0,APO_FAC 50.0,AXIS_VEL 100.0,AXIS_ACC 100.0,ORI_TYP #VAR,CIRC_TYP #BASE,JERK_FAC 50.0,GEAR_JERK 50.0,EXAX_IGN 0}
DECL LDAT LCPDAT11={VEL 2.0,ACC 100.0,APO_DIST 30.0,APO_FAC 50.0,AXIS_VEL 100.0,AXIS_ACC 100.0,ORI_TYP #VAR,CIRC_TYP #BASE,JERK_FAC 50.0,GEAR_JERK 50.0,EXAX_IGN 0}
DECL SPOT_SUGG_T LAST_SPOT={GUN[] "2                       ",RETR_CMD[] "#CLO                    ",CHOISE[] "#FIRST                  ",CLO_TM[] "1                       ",PGNO1[] "186                     ",PRESS1[] "0                       ",PGNO2[] "1                       ",PRESS2[] "0                       ",SPOT_PARAMS[] "NORMAL                  "}
DECL E6POS XP13={X 1734.21204,Y -1867.81604,Z 844.310181,A 176.924194,B -49.5563011,C -94.5412521,S 18,T 11,E1 0.0,E2 0.0,E3 0.0,E4 0.0,E5 0.0,E6 0.0}
DECL FDAT FP13={TOOL_NO 3,BASE_NO 3,IPO_FRAME #BASE,POINT2[] " ",TQ_STATE FALSE}
DECL PDAT PPDAT10={VEL 100.0,ACC 80.0,APO_DIST 100.0,APO_MODE #CDIS,GEAR_JERK 50.0}
DECL PDAT PP_OLP7={VEL 100.0,ACC 100.0,APO_DIST 0.0}
DECL E6POS Xl007={X 1644.52502,Y -2192.26294,Z 368.696686,A 170.023499,B -52.7817612,C -87.1773682,S 18,T 3,E1 0.0,E2 0.0,E3 0.0,E4 0.0,E5 0.0,E6 0.0}
DECL FDAT Fl007={TOOL_NO 3,BASE_NO 3,IPO_FRAME #BASE,POINT2[] " "}
DECL PDAT PP_OLP8={VEL 100.0,ACC 100.0,APO_DIST 30.0,APO_MODE #CDIS}
DECL E6POS Xl008={X 745.877075,Y -1613.48499,Z 78.2501373,A -16.3194294,B 12.0206604,C -22.6783009,S 18,T 3,E1 0.0,E2 0.0,E3 0.0,E4 0.0,E5 0.0,E6 0.0}
DECL FDAT Fl008={TOOL_NO 3,BASE_NO 3,IPO_FRAME #BASE,POINT2[] " "}
DECL LDAT LL_OLP65={VEL 2.0,ACC 100.0,APO_DIST 10.0,APO_FAC 0.0,ORI_TYP #VAR,CIRC_TYP #BASE,JERK_FAC 50.0}
DECL E6POS Xl042={X 120.267197,Y -792.371704,Z 628.356201,A -114.714401,B 75.1284332,C -117.9123,S 18,T 35,E1 0.0,E2 0.0,E3 0.0,E4 0.0,E5 0.0,E6 0.0}
DECL FDAT Fl042={TOOL_NO 3,BASE_NO 3,IPO_FRAME #BASE,POINT2[] " "}
DECL E6POS XSWP_60_7345={X 142.078003,Y -899.095581,Z 596.340515,A -114.726898,B 75.1311569,C -119.781998,S 18,T 35,E1 0.0,E2 0.0,E3 0.0,E4 0.0,E5 0.0,E6 0.0}
DECL FDAT FSWP_60_7345={TOOL_NO 3,BASE_NO 3,IPO_FRAME #BASE,POINT2[] " "}
DECL E6POS XSWP_60_7897={X 107.698997,Y -641.672424,Z 593.484924,A -111.071098,B 80.2933578,C -110.974403,S 18,T 35,E1 0.0,E2 0.0,E3 0.0,E4 0.0,E5 0.0,E6 0.0}
DECL FDAT FSWP_60_7897={TOOL_NO 3,BASE_NO 3,IPO_FRAME #BASE,POINT2[] " "}
DECL E6POS XSWP_60_7311={X 92.3604965,Y -351.341614,Z 592.924377,A -131.178406,B 80.0360565,C -134.013107,S 18,T 35,E1 0.0,E2 0.0,E3 0.0,E4 0.0,E5 0.0,E6 0.0}
DECL FDAT FSWP_60_7311={TOOL_NO 3,BASE_NO 3,IPO_FRAME #BASE,POINT2[] " "}
DECL LDAT LCPDAT13={VEL 2.0,ACC 100.0,APO_DIST 100.0,APO_FAC 50.0,AXIS_VEL 100.0,AXIS_ACC 100.0,ORI_TYP #VAR,CIRC_TYP #BASE,JERK_FAC 50.0,GEAR_JERK 50.0,EXAX_IGN 0}
DECL LDAT LCPDAT14={VEL 2.0,ACC 100.0,APO_DIST 100.0,APO_FAC 50.0,AXIS_VEL 100.0,AXIS_ACC 100.0,ORI_TYP #VAR,CIRC_TYP #BASE,JERK_FAC 50.0,GEAR_JERK 50.0,EXAX_IGN 0}
DECL LDAT LCPDAT15={VEL 2.0,ACC 90.0,APO_DIST 5.0,APO_FAC 50.0,AXIS_VEL 100.0,AXIS_ACC 100.0,ORI_TYP #VAR,CIRC_TYP #BASE,JERK_FAC 50.0,GEAR_JERK 50.0,EXAX_IGN 0}
DECL E6POS XP15={X 1113.95496,Y -991.188293,Z 14.3488798,A 179.752701,B -16.1354008,C -89.9455795,S 18,T 43,E1 0.0,E2 0.0,E3 0.0,E4 0.0,E5 0.0,E6 0.0}
DECL FDAT FP15={TOOL_NO 3,BASE_NO 3,IPO_FRAME #BASE,POINT2[] " ",TQ_STATE FALSE}
DECL LDAT LCPDAT16={VEL 2.0,ACC 100.0,APO_DIST 5.0,APO_FAC 50.0,AXIS_VEL 100.0,AXIS_ACC 100.0,ORI_TYP #VAR,CIRC_TYP #BASE,JERK_FAC 50.0,GEAR_JERK 50.0,EXAX_IGN 0}
DECL E6POS XP16={X 1106.151,Y -1003.31702,Z 67.7898407,A 179.753098,B -16.1340904,C -89.9462967,S 18,T 43,E1 0.0,E2 0.0,E3 0.0,E4 0.0,E5 0.0,E6 0.0}
DECL FDAT FP16={TOOL_NO 3,BASE_NO 3,IPO_FRAME #BASE,POINT2[] " ",TQ_STATE FALSE}
DECL LDAT LCPDAT17={VEL 2.0,ACC 100.0,APO_DIST 100.0,APO_FAC 50.0,AXIS_VEL 100.0,AXIS_ACC 100.0,ORI_TYP #VAR,CIRC_TYP #BASE,JERK_FAC 50.0,GEAR_JERK 50.0,EXAX_IGN 0}
DECL E6POS XSWP_61_7027={X 1112.39697,Y -1015.453,Z 71.4506226,A 179.753098,B -16.1340103,C -89.9465027,S 18,T 43,E1 0.0,E2 0.0,E3 0.0,E4 0.0,E5 0.0,E6 0.0}
DECL FDAT FSWP_61_7027={TOOL_NO 3,BASE_NO 3,IPO_FRAME #BASE,POINT2[] " ",TQ_STATE FALSE}
DECL LDAT LCPDAT18={VEL 2.0,ACC 100.0,APO_DIST 100.0,APO_FAC 50.0,AXIS_VEL 100.0,AXIS_ACC 100.0,ORI_TYP #VAR,CIRC_TYP #BASE,JERK_FAC 50.0,GEAR_JERK 50.0,EXAX_IGN 0}
DECL E6POS XSWP_61_7029={X 1176.19299,Y -1021.13898,Z 95.2776031,A 179.752304,B -16.1331501,C -89.9456406,S 18,T 43,E1 0.0,E2 0.0,E3 0.0,E4 0.0,E5 0.0,E6 0.0}
DECL FDAT FSWP_61_7029={TOOL_NO 3,BASE_NO 3,IPO_FRAME #BASE,POINT2[] " ",TQ_STATE FALSE}
DECL LDAT LCPDAT19={VEL 2.0,ACC 100.0,APO_DIST 100.0,APO_FAC 50.0,AXIS_VEL 100.0,AXIS_ACC 100.0,ORI_TYP #VAR,CIRC_TYP #BASE,JERK_FAC 50.0,GEAR_JERK 50.0,EXAX_IGN 0}
DECL E6POS XSWP_61_7031={X 1228.125,Y -1021.565,Z 105.6548,A 179.7388,B -30.3301392,C -89.944603,S 18,T 43,E1 0.0,E2 0.0,E3 0.0,E4 0.0,E5 0.0,E6 0.0}
DECL FDAT FSWP_61_7031={TOOL_NO 3,BASE_NO 3,IPO_FRAME #BASE,POINT2[] " ",TQ_STATE FALSE}
DECL E6POS XP17={X 1220.47095,Y -1002.95001,Z 54.8409309,A 179.738998,B -30.3312206,C -89.9440231,S 18,T 43,E1 0.0,E2 0.0,E3 0.0,E4 0.0,E5 0.0,E6 0.0}
DECL FDAT FP17={TOOL_NO 3,BASE_NO 3,IPO_FRAME #BASE,POINT2[] " ",TQ_STATE FALSE}
DECL LDAT LCPDAT21={VEL 2.0,ACC 100.0,APO_DIST 150.0,APO_FAC 50.0,AXIS_VEL 100.0,AXIS_ACC 100.0,ORI_TYP #VAR,CIRC_TYP #BASE,JERK_FAC 50.0,GEAR_JERK 50.0,EXAX_IGN 0}
DECL PDAT PPDAT13={VEL 100.0,ACC 100.0,APO_DIST 100.0,APO_MODE #CDIS,GEAR_JERK 50.0}
DECL E6POS XP18={X 1384.60303,Y -1894.59204,Z 1393.06104,A -86.6525192,B -54.8740196,C 168.649399,S 22,T 19,E1 0.0,E2 0.0,E3 0.0,E4 0.0,E5 0.0,E6 0.0}
DECL FDAT FP18={TOOL_NO 3,BASE_NO 3,IPO_FRAME #BASE,POINT2[] " ",TQ_STATE FALSE}
DECL LDAT LCPDAT23={VEL 2.0,ACC 100.0,APO_DIST 150.0,APO_FAC 50.0,AXIS_VEL 100.0,AXIS_ACC 100.0,ORI_TYP #VAR,CIRC_TYP #BASE,JERK_FAC 50.0,GEAR_JERK 50.0,EXAX_IGN 0}
ENDDAT
